ABB RAPID module: P41.mod

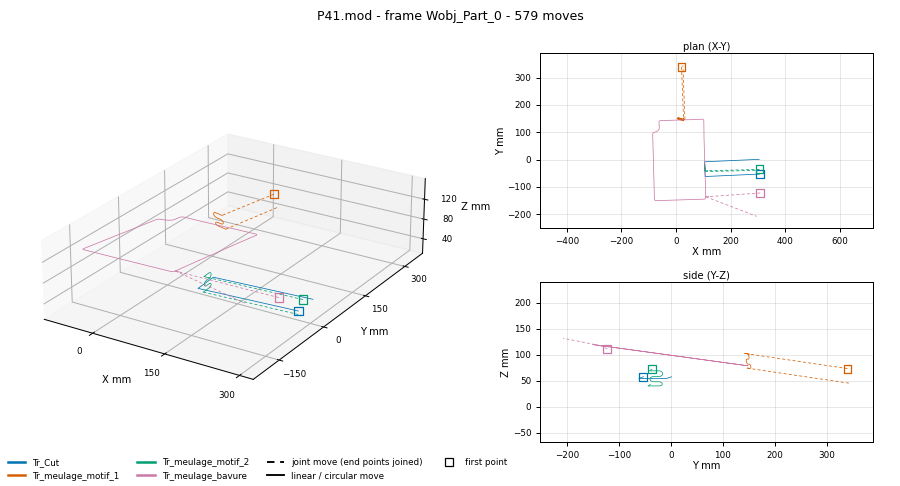
[picture p0: tool path of P41.mod in frame Wobj_Part_0, 579 of 588 moves have a stored position in this frame; points joined in program order, loops and branches not executed]
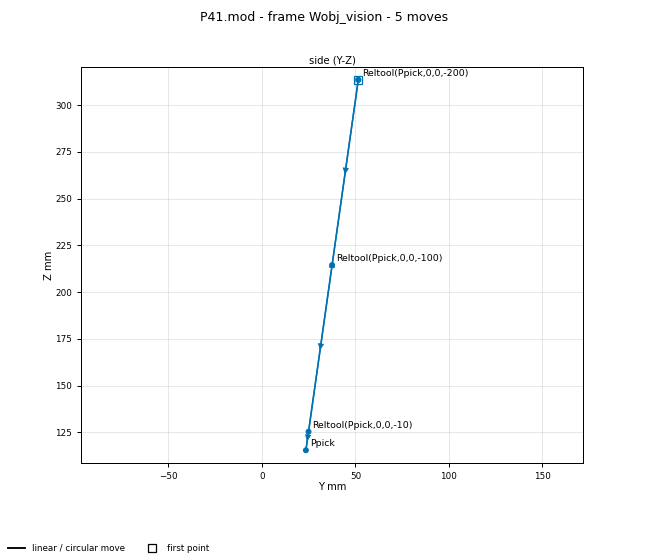
[picture p1: tool path of P41.mod in frame Wobj_vision, 5 of 588 moves have a stored position in this frame; points joined in program order, loops and branches not executed]
MODULE P41
	LOCAL CONST Speeddata vitesse_Tronconnage :=[10, 500, 0, 0];
	LOCAL CONST Robtarget Coupe_0 :=[[105.2163046875,-29.7869296875,54.5294296875],[0.0104555272873827,0.0212605825828778,-0.706787087904297,-0.707029477425901],[0,0,0,0],[8.999999E+09,8.999999E+09,8.999999E+09,8.999999E+09,8.999999E+09,8.999999E+09]];
	LOCAL CONST Robtarget Tr_meulage_motif_1_App1 :=[[20.0512236789454,339.562295836737,73.4032374615753],[0.0144291641931026,-0.0124615274841837,0.653500364086891,-0.756686053586129],[0,0,0,0],[8.999999E+09,8.999999E+09,8.999999E+09,8.999999E+09,8.999999E+09,8.999999E+09]];
	LOCAL CONST Robtarget Tr_meulage_motif_1_App2 :=[[27.2176163597285,151.722671041837,101.060391560579],[0.0144291641931026,-0.0124615274841837,0.653500364086891,-0.756686053586129],[0,0,0,0],[8.999999E+09,8.999999E+09,8.999999E+09,8.999999E+09,8.999999E+09,8.999999E+09]];
	LOCAL CONST Robtarget Tr_meulage_motif_1_P0 :=[[27.594794921875,141.836375,102.51603125],[0.0144291641931026,-0.0124615274841837,0.653500364086891,-0.756686053586129],[0,0,0,0],[8.999999E+09,8.999999E+09,8.999999E+09,8.999999E+09,8.999999E+09,8.999999E+09]];
	LOCAL CONST Robtarget Tr_meulage_motif_1_P1 :=[[26.6349609375,142.116578125,102.5018671875],[0.0144291641931026,-0.0124615274841837,0.653500364086891,-0.756686053586129],[0,0,0,0],[8.999999E+09,8.999999E+09,8.999999E+09,8.999999E+09,8.999999E+09,8.999999E+09]];
	LOCAL CONST Robtarget Tr_meulage_motif_1_P2 :=[[25.675126953125,142.396796875,102.487703125],[0.0144291641931026,-0.0124615274841837,0.653500364086891,-0.756686053586129],[0,0,0,0],[8.999999E+09,8.999999E+09,8.999999E+09,8.999999E+09,8.999999E+09,8.999999E+09]];
	LOCAL CONST Robtarget Tr_meulage_motif_1_P3 :=[[24.71529296875,142.677,102.4735390625],[0.0144291641931026,-0.0124615274841837,0.653500364086891,-0.756686053586129],[0,0,0,0],[8.999999E+09,8.999999E+09,8.999999E+09,8.999999E+09,8.999999E+09,8.999999E+09]];
	LOCAL CONST Robtarget Tr_meulage_motif_1_P4 :=[[23.755458984375,142.95721875,102.4593671875],[0.0144291641931026,-0.0124615274841837,0.653500364086891,-0.756686053586129],[0,0,0,0],[8.999999E+09,8.999999E+09,8.999999E+09,8.999999E+09,8.999999E+09,8.999999E+09]];
	LOCAL CONST Robtarget Tr_meulage_motif_1_P5 :=[[22.795625,143.237421875,102.445203125],[0.0144291641931026,-0.0124615274841837,0.653500364086891,-0.756686053586129],[0,0,0,0],[8.999999E+09,8.999999E+09,8.999999E+09,8.999999E+09,8.999999E+09,8.999999E+09]];
	LOCAL CONST Robtarget Tr_meulage_motif_1_P6 :=[[21.835791015625,143.517640625,102.4310390625],[0.0144291641931026,-0.0124615274841837,0.653500364086891,-0.756686053586129],[0,0,0,0],[8.999999E+09,8.999999E+09,8.999999E+09,8.999999E+09,8.999999E+09,8.999999E+09]];
	LOCAL CONST Robtarget Tr_meulage_motif_1_P7 :=[[20.87595703125,143.79784375,102.416875],[0.0144291641931026,-0.0124615274841837,0.653500364086891,-0.756686053586129],[0,0,0,0],[8.999999E+09,8.999999E+09,8.999999E+09,8.999999E+09,8.999999E+09,8.999999E+09]];
	LOCAL CONST Robtarget Tr_meulage_motif_1_P8 :=[[19.916123046875,144.0780625,102.4027109375],[0.0144291641931026,-0.0124615274841837,0.653500364086891,-0.756686053586129],[0,0,0,0],[8.999999E+09,8.999999E+09,8.999999E+09,8.999999E+09,8.999999E+09,8.999999E+09]];
	LOCAL CONST Robtarget Tr_meulage_motif_1_P9 :=[[18.9562890625,144.358265625,102.3885390625],[0.0144291641931026,-0.0124615274841837,0.653500364086891,-0.756686053586129],[0,0,0,0],[8.999999E+09,8.999999E+09,8.999999E+09,8.999999E+09,8.999999E+09,8.999999E+09]];
	LOCAL CONST Robtarget Tr_meulage_motif_1_P10 :=[[17.99645703125,144.638484375,102.374375],[0.0144291641931026,-0.0124615274841837,0.653500364086891,-0.756686053586129],[0,0,0,0],[8.999999E+09,8.999999E+09,8.999999E+09,8.999999E+09,8.999999E+09,8.999999E+09]];
	LOCAL CONST Robtarget Tr_meulage_motif_1_P11 :=[[17.036623046875,144.9186875,102.3602109375],[0.0144291641931026,-0.0124615274841837,0.653500364086891,-0.756686053586129],[0,0,0,0],[8.999999E+09,8.999999E+09,8.999999E+09,8.999999E+09,8.999999E+09,8.999999E+09]];
	LOCAL CONST Robtarget Tr_meulage_motif_1_P12 :=[[16.0767880859375,145.19890625,102.346046875],[0.0144291641931026,-0.0124615274841837,0.653500364086891,-0.756686053586129],[0,0,0,0],[8.999999E+09,8.999999E+09,8.999999E+09,8.999999E+09,8.999999E+09,8.999999E+09]];
	LOCAL CONST Robtarget Tr_meulage_motif_1_P13 :=[[15.116955078125,145.479109375,102.331875],[0.0144291641931026,-0.0124615274841837,0.653500364086891,-0.756686053586129],[0,0,0,0],[8.999999E+09,8.999999E+09,8.999999E+09,8.999999E+09,8.999999E+09,8.999999E+09]];
	LOCAL CONST Robtarget Tr_meulage_motif_1_P14 :=[[14.15712109375,145.759328125,102.3177109375],[0.0144291641931026,-0.0124615274841837,0.653500364086891,-0.756686053586129],[0,0,0,0],[8.999999E+09,8.999999E+09,8.999999E+09,8.999999E+09,8.999999E+09,8.999999E+09]];
	LOCAL CONST Robtarget Tr_meulage_motif_1_P15 :=[[13.197287109375,146.03953125,102.303546875],[0.0144291641931026,-0.0124615274841837,0.653500364086891,-0.756686053586129],[0,0,0,0],[8.999999E+09,8.999999E+09,8.999999E+09,8.999999E+09,8.999999E+09,8.999999E+09]];
	LOCAL CONST Robtarget Tr_meulage_motif_1_P16 :=[[12.237453125,146.31975,102.2893828125],[0.0144291641931026,-0.0124615274841837,0.653500364086891,-0.756686053586129],[0,0,0,0],[8.999999E+09,8.999999E+09,8.999999E+09,8.999999E+09,8.999999E+09,8.999999E+09]];
	LOCAL CONST Robtarget Tr_meulage_motif_1_P17 :=[[11.277619140625,146.59996875,102.27521875],[0.0144291641931026,-0.0124615274841837,0.653500364086891,-0.756686053586129],[0,0,0,0],[8.999999E+09,8.999999E+09,8.999999E+09,8.999999E+09,8.999999E+09,8.999999E+09]];
	LOCAL CONST Robtarget Tr_meulage_motif_1_P18 :=[[10.31778515625,146.880171875,102.261046875],[0.0144291641931026,-0.0124615274841837,0.653500364086891,-0.756686053586129],[0,0,0,0],[8.999999E+09,8.999999E+09,8.999999E+09,8.999999E+09,8.999999E+09,8.999999E+09]];
	LOCAL CONST Robtarget Tr_meulage_motif_1_P19 :=[[9.3730380859375,147.1800625,102.1388515625],[0.0144291641931026,-0.0124615274841837,0.653500364086891,-0.756686053586129],[0,0,0,0],[8.999999E+09,8.999999E+09,8.999999E+09,8.999999E+09,8.999999E+09,8.999999E+09]];
	LOCAL CONST Robtarget Tr_meulage_motif_1_P20 :=[[8.4797333984375,147.486828125,101.9189375],[0.0144291641931026,-0.0124615274841837,0.653500364086891,-0.756686053586129],[0,0,0,0],[8.999999E+09,8.999999E+09,8.999999E+09,8.999999E+09,8.999999E+09,8.999999E+09]];
	LOCAL CONST Robtarget Tr_meulage_motif_1_P21 :=[[7.68080224609375,147.77925,101.641046875],[0.0144291641931026,-0.0124615274841837,0.653500364086891,-0.756686053586129],[0,0,0,0],[8.999999E+09,8.999999E+09,8.999999E+09,8.999999E+09,8.999999E+09,8.999999E+09]];
	LOCAL CONST Robtarget Tr_meulage_motif_1_P22 :=[[6.98081787109375,148.0436875,101.3606015625],[0.0144291641931026,-0.0124615274841837,0.653500364086891,-0.756686053586129],[0,0,0,0],[8.999999E+09,8.999999E+09,8.999999E+09,8.999999E+09,8.999999E+09,8.999999E+09]];
	LOCAL CONST Robtarget Tr_meulage_motif_1_P23 :=[[5.96826025390625,148.4734375,100.742546875],[0.0144291641931026,-0.0124615274841837,0.653500364086891,-0.756686053586129],[0,0,0,0],[8.999999E+09,8.999999E+09,8.999999E+09,8.999999E+09,8.999999E+09,8.999999E+09]];
	LOCAL CONST Robtarget Tr_meulage_motif_1_P24 :=[[5.0464296875,148.927109375,99.8991953125],[0.0144291641931026,-0.0124615274841837,0.653500364086891,-0.756686053586129],[0,0,0,0],[8.999999E+09,8.999999E+09,8.999999E+09,8.999999E+09,8.999999E+09,8.999999E+09]];
	LOCAL CONST Robtarget Tr_meulage_motif_1_P25 :=[[4.30640478515625,149.3660625,98.8860234375],[0.0144291641931026,-0.0124615274841837,0.653500364086891,-0.756686053586129],[0,0,0,0],[8.999999E+09,8.999999E+09,8.999999E+09,8.999999E+09,8.999999E+09,8.999999E+09]];
	LOCAL CONST Robtarget Tr_meulage_motif_1_P26 :=[[3.91807373046875,149.722453125,97.7876796875],[0.0144291641931026,-0.0124615274841837,0.653500364086891,-0.756686053586129],[0,0,0,0],[8.999999E+09,8.999999E+09,8.999999E+09,8.999999E+09,8.999999E+09,8.999999E+09]];
	LOCAL CONST Robtarget Tr_meulage_motif_1_P27 :=[[3.9421162109375,149.86696875,97.106765625],[0.0144291641931026,-0.0124615274841837,0.653500364086891,-0.756686053586129],[0,0,0,0],[8.999999E+09,8.999999E+09,8.999999E+09,8.999999E+09,8.999999E+09,8.999999E+09]];
	LOCAL CONST Robtarget Tr_meulage_motif_1_P28 :=[[3.98963891601562,149.9970625,96.4601875],[0.0144291641931026,-0.0124615274841837,0.653500364086891,-0.756686053586129],[0,0,0,0],[8.999999E+09,8.999999E+09,8.999999E+09,8.999999E+09,8.999999E+09,8.999999E+09]];
	LOCAL CONST Robtarget Tr_meulage_motif_1_P29 :=[[4.0898212890625,150.11175,95.81453125],[0.0144291641931026,-0.0124615274841837,0.653500364086891,-0.756686053586129],[0,0,0,0],[8.999999E+09,8.999999E+09,8.999999E+09,8.999999E+09,8.999999E+09,8.999999E+09]];
	LOCAL CONST Robtarget Tr_meulage_motif_1_P30 :=[[4.647208984375,150.18890625,94.74428125],[0.0144291641931026,-0.0124615274841837,0.653500364086891,-0.756686053586129],[0,0,0,0],[8.999999E+09,8.999999E+09,8.999999E+09,8.999999E+09,8.999999E+09,8.999999E+09]];
	LOCAL CONST Robtarget Tr_meulage_motif_1_P31 :=[[5.54177099609375,150.146921875,93.7721171875],[0.0144291641931026,-0.0124615274841837,0.653500364086891,-0.756686053586129],[0,0,0,0],[8.999999E+09,8.999999E+09,8.999999E+09,8.999999E+09,8.999999E+09,8.999999E+09]];
	LOCAL CONST Robtarget Tr_meulage_motif_1_P32 :=[[6.583640625,150.023234375,92.976125],[0.0144291641931026,-0.0124615274841837,0.653500364086891,-0.756686053586129],[0,0,0,0],[8.999999E+09,8.999999E+09,8.999999E+09,8.999999E+09,8.999999E+09,8.999999E+09]];
	LOCAL CONST Robtarget Tr_meulage_motif_1_P33 :=[[7.271578125,149.9085625,92.598890625],[0.0144291641931026,-0.0124615274841837,0.653500364086891,-0.756686053586129],[0,0,0,0],[8.999999E+09,8.999999E+09,8.999999E+09,8.999999E+09,8.999999E+09,8.999999E+09]];
	LOCAL CONST Robtarget Tr_meulage_motif_1_P34 :=[[8.41825390625,149.679953125,92.138578125],[0.0144291641931026,-0.0124615274841837,0.653500364086891,-0.756686053586129],[0,0,0,0],[8.999999E+09,8.999999E+09,8.999999E+09,8.999999E+09,8.999999E+09,8.999999E+09]];
	LOCAL CONST Robtarget Tr_meulage_motif_1_P35 :=[[9.2483232421875,149.495125,91.8923125],[0.0144291641931026,-0.0124615274841837,0.653500364086891,-0.756686053586129],[0,0,0,0],[8.999999E+09,8.999999E+09,8.999999E+09,8.999999E+09,8.999999E+09,8.999999E+09]];
	LOCAL CONST Robtarget Tr_meulage_motif_1_P36 :=[[10.1575830078125,149.2741875,91.7055859375],[0.0144291641931026,-0.0124615274841837,0.653500364086891,-0.756686053586129],[0,0,0,0],[8.999999E+09,8.999999E+09,8.999999E+09,8.999999E+09,8.999999E+09,8.999999E+09]];
	LOCAL CONST Robtarget Tr_meulage_motif_1_P37 :=[[11.1075244140625,149.020515625,91.6133046875],[0.0144291641931026,-0.0124615274841837,0.653500364086891,-0.756686053586129],[0,0,0,0],[8.999999E+09,8.999999E+09,8.999999E+09,8.999999E+09,8.999999E+09,8.999999E+09]];
	LOCAL CONST Robtarget Tr_meulage_motif_1_P38 :=[[12.0681669921875,148.764140625,91.5192265625],[0.0144291641931026,-0.0124615274841837,0.653500364086891,-0.756686053586129],[0,0,0,0],[8.999999E+09,8.999999E+09,8.999999E+09,8.999999E+09,8.999999E+09,8.999999E+09]];
	LOCAL CONST Robtarget Tr_meulage_motif_1_P39 :=[[13.0280009765625,148.4839375,91.533390625],[0.0144291641931026,-0.0124615274841837,0.653500364086891,-0.756686053586129],[0,0,0,0],[8.999999E+09,8.999999E+09,8.999999E+09,8.999999E+09,8.999999E+09,8.999999E+09]];
	LOCAL CONST Robtarget Tr_meulage_motif_1_P40 :=[[13.9878349609375,148.20371875,91.5475546875],[0.0144291641931026,-0.0124615274841837,0.653500364086891,-0.756686053586129],[0,0,0,0],[8.999999E+09,8.999999E+09,8.999999E+09,8.999999E+09,8.999999E+09,8.999999E+09]];
	LOCAL CONST Robtarget Tr_meulage_motif_1_P41 :=[[14.9476689453125,147.9235,91.56171875],[0.0144291641931026,-0.0124615274841837,0.653500364086891,-0.756686053586129],[0,0,0,0],[8.999999E+09,8.999999E+09,8.999999E+09,8.999999E+09,8.999999E+09,8.999999E+09]];
	LOCAL CONST Robtarget Tr_meulage_motif_1_P42 :=[[15.9075029296875,147.643296875,91.575890625],[0.0144291641931026,-0.0124615274841837,0.653500364086891,-0.756686053586129],[0,0,0,0],[8.999999E+09,8.999999E+09,8.999999E+09,8.999999E+09,8.999999E+09,8.999999E+09]];
	LOCAL CONST Robtarget Tr_meulage_motif_1_P43 :=[[16.8673359375,147.363078125,91.5900546875],[0.0144291641931026,-0.0124615274841837,0.653500364086891,-0.756686053586129],[0,0,0,0],[8.999999E+09,8.999999E+09,8.999999E+09,8.999999E+09,8.999999E+09,8.999999E+09]];
	LOCAL CONST Robtarget Tr_meulage_motif_1_P44 :=[[17.827169921875,147.082875,91.60421875],[0.0144291641931026,-0.0124615274841837,0.653500364086891,-0.756686053586129],[0,0,0,0],[8.999999E+09,8.999999E+09,8.999999E+09,8.999999E+09,8.999999E+09,8.999999E+09]];
	LOCAL CONST Robtarget Tr_meulage_motif_1_P45 :=[[18.78700390625,146.80265625,91.6183828125],[0.0144291641931026,-0.0124615274841837,0.653500364086891,-0.756686053586129],[0,0,0,0],[8.999999E+09,8.999999E+09,8.999999E+09,8.999999E+09,8.999999E+09,8.999999E+09]];
	LOCAL CONST Robtarget Tr_meulage_motif_1_P46 :=[[19.746837890625,146.522453125,91.632546875],[0.0144291641931026,-0.0124615274841837,0.653500364086891,-0.756686053586129],[0,0,0,0],[8.999999E+09,8.999999E+09,8.999999E+09,8.999999E+09,8.999999E+09,8.999999E+09]];
	LOCAL CONST Robtarget Tr_meulage_motif_1_P47 :=[[20.706671875,146.242234375,91.64671875],[0.0144291641931026,-0.0124615274841837,0.653500364086891,-0.756686053586129],[0,0,0,0],[8.999999E+09,8.999999E+09,8.999999E+09,8.999999E+09,8.999999E+09,8.999999E+09]];
	LOCAL CONST Robtarget Tr_meulage_motif_1_P48 :=[[21.666505859375,145.96203125,91.6608828125],[0.0144291641931026,-0.0124615274841837,0.653500364086891,-0.756686053586129],[0,0,0,0],[8.999999E+09,8.999999E+09,8.999999E+09,8.999999E+09,8.999999E+09,8.999999E+09]];
	LOCAL CONST Robtarget Tr_meulage_motif_1_P49 :=[[22.6271484375,145.70565625,91.5668046875],[0.0144291641931026,-0.0124615274841837,0.653500364086891,-0.756686053586129],[0,0,0,0],[8.999999E+09,8.999999E+09,8.999999E+09,8.999999E+09,8.999999E+09,8.999999E+09]];
	LOCAL CONST Robtarget Tr_meulage_motif_1_P50 :=[[23.55080859375,145.481984375,91.373703125],[0.0144291641931026,-0.0124615274841837,0.653500364086891,-0.756686053586129],[0,0,0,0],[8.999999E+09,8.999999E+09,8.999999E+09,8.999999E+09,8.999999E+09,8.999999E+09]];
	LOCAL CONST Robtarget Tr_meulage_motif_1_P51 :=[[24.388814453125,145.29653125,91.11996875],[0.0144291641931026,-0.0124615274841837,0.653500364086891,-0.756686053586129],[0,0,0,0],[8.999999E+09,8.999999E+09,8.999999E+09,8.999999E+09,8.999999E+09,8.999999E+09]];
	LOCAL CONST Robtarget Tr_meulage_motif_1_P52 :=[[25.093595703125,145.157,90.832640625],[0.0144291641931026,-0.0124615274841837,0.653500364086891,-0.756686053586129],[0,0,0,0],[8.999999E+09,8.999999E+09,8.999999E+09,8.999999E+09,8.999999E+09,8.999999E+09]];
	LOCAL CONST Robtarget Tr_meulage_motif_1_P53 :=[[26.13412890625,144.997484375,90.1994609375],[0.0144291641931026,-0.0124615274841837,0.653500364086891,-0.756686053586129],[0,0,0,0],[8.999999E+09,8.999999E+09,8.999999E+09,8.999999E+09,8.999999E+09,8.999999E+09]];
	LOCAL CONST Robtarget Tr_meulage_motif_1_P54 :=[[27.064658203125,144.922203125,89.3303046875],[0.0144291641931026,-0.0124615274841837,0.653500364086891,-0.756686053586129],[0,0,0,0],[8.999999E+09,8.999999E+09,8.999999E+09,8.999999E+09,8.999999E+09,8.999999E+09]];
	LOCAL CONST Robtarget Tr_meulage_motif_1_P55 :=[[27.65331640625,144.97809375,88.3150625],[0.0144291641931026,-0.0124615274841837,0.653500364086891,-0.756686053586129],[0,0,0,0],[8.999999E+09,8.999999E+09,8.999999E+09,8.999999E+09,8.999999E+09,8.999999E+09]];
	LOCAL CONST Robtarget Tr_meulage_motif_1_P56 :=[[27.88049609375,145.062703125,87.6398359375],[0.0144291641931026,-0.0124615274841837,0.653500364086891,-0.756686053586129],[0,0,0,0],[8.999999E+09,8.999999E+09,8.999999E+09,8.999999E+09,8.999999E+09,8.999999E+09]];
	LOCAL CONST Robtarget Tr_meulage_motif_1_P57 :=[[27.99711328125,145.1963125,86.8878203125],[0.0144291641931026,-0.0124615274841837,0.653500364086891,-0.756686053586129],[0,0,0,0],[8.999999E+09,8.999999E+09,8.999999E+09,8.999999E+09,8.999999E+09,8.999999E+09]];
	LOCAL CONST Robtarget Tr_meulage_motif_1_P58 :=[[27.988193359375,145.36653125,86.134078125],[0.0144291641931026,-0.0124615274841837,0.653500364086891,-0.756686053586129],[0,0,0,0],[8.999999E+09,8.999999E+09,8.999999E+09,8.999999E+09,8.999999E+09,8.999999E+09]];
	LOCAL CONST Robtarget Tr_meulage_motif_1_P59 :=[[27.6651015625,145.702140625,85.0444609375],[0.0144291641931026,-0.0124615274841837,0.653500364086891,-0.756686053586129],[0,0,0,0],[8.999999E+09,8.999999E+09,8.999999E+09,8.999999E+09,8.999999E+09,8.999999E+09]];
	LOCAL CONST Robtarget Tr_meulage_motif_1_P60 :=[[27.309521484375,145.93346875,84.4658984375],[0.0144291641931026,-0.0124615274841837,0.653500364086891,-0.756686053586129],[0,0,0,0],[8.999999E+09,8.999999E+09,8.999999E+09,8.999999E+09,8.999999E+09,8.999999E+09]];
	LOCAL CONST Robtarget Tr_meulage_motif_1_P61 :=[[26.52178515625,146.35659375,83.585890625],[0.0144291641931026,-0.0124615274841837,0.653500364086891,-0.756686053586129],[0,0,0,0],[8.999999E+09,8.999999E+09,8.999999E+09,8.999999E+09,8.999999E+09,8.999999E+09]];
	LOCAL CONST Robtarget Tr_meulage_motif_1_P62 :=[[25.9893984375,146.60221875,83.17246875],[0.0144291641931026,-0.0124615274841837,0.653500364086891,-0.756686053586129],[0,0,0,0],[8.999999E+09,8.999999E+09,8.999999E+09,8.999999E+09,8.999999E+09,8.999999E+09]];
	LOCAL CONST Robtarget Tr_meulage_motif_1_P63 :=[[24.955498046875,147.022515625,82.624609375],[0.0144291641931026,-0.0124615274841837,0.653500364086891,-0.756686053586129],[0,0,0,0],[8.999999E+09,8.999999E+09,8.999999E+09,8.999999E+09,8.999999E+09,8.999999E+09]];
	LOCAL CONST Robtarget Tr_meulage_motif_1_P64 :=[[24.18430078125,147.312,82.32396875],[0.0144291641931026,-0.0124615274841837,0.653500364086891,-0.756686053586129],[0,0,0,0],[8.999999E+09,8.999999E+09,8.999999E+09,8.999999E+09,8.999999E+09,8.999999E+09]];
	LOCAL CONST Robtarget Tr_meulage_motif_1_P65 :=[[23.304431640625,147.613375,82.110828125],[0.0144291641931026,-0.0124615274841837,0.653500364086891,-0.756686053586129],[0,0,0,0],[8.999999E+09,8.999999E+09,8.999999E+09,8.999999E+09,8.999999E+09,8.999999E+09]];
	LOCAL CONST Robtarget Tr_meulage_motif_1_P66 :=[[22.370099609375,147.909796875,81.9907421875],[0.0144291641931026,-0.0124615274841837,0.653500364086891,-0.756686053586129],[0,0,0,0],[8.999999E+09,8.999999E+09,8.999999E+09,8.999999E+09,8.999999E+09,8.999999E+09]];
	LOCAL CONST Robtarget Tr_meulage_motif_1_P67 :=[[21.4253515625,148.209671875,81.8685390625],[0.0144291641931026,-0.0124615274841837,0.653500364086891,-0.756686053586129],[0,0,0,0],[8.999999E+09,8.999999E+09,8.999999E+09,8.999999E+09,8.999999E+09,8.999999E+09]];
	LOCAL CONST Robtarget Tr_meulage_motif_1_P68 :=[[20.465517578125,148.489890625,81.854375],[0.0144291641931026,-0.0124615274841837,0.653500364086891,-0.756686053586129],[0,0,0,0],[8.999999E+09,8.999999E+09,8.999999E+09,8.999999E+09,8.999999E+09,8.999999E+09]];
	LOCAL CONST Robtarget Tr_meulage_motif_1_P69 :=[[19.50568359375,148.77009375,81.8402109375],[0.0144291641931026,-0.0124615274841837,0.653500364086891,-0.756686053586129],[0,0,0,0],[8.999999E+09,8.999999E+09,8.999999E+09,8.999999E+09,8.999999E+09,8.999999E+09]];
	LOCAL CONST Robtarget Tr_meulage_motif_1_P70 :=[[18.545849609375,149.0503125,81.826046875],[0.0144291641931026,-0.0124615274841837,0.653500364086891,-0.756686053586129],[0,0,0,0],[8.999999E+09,8.999999E+09,8.999999E+09,8.999999E+09,8.999999E+09,8.999999E+09]];
	LOCAL CONST Robtarget Tr_meulage_motif_1_P71 :=[[17.586015625,149.330515625,81.811875],[0.0144291641931026,-0.0124615274841837,0.653500364086891,-0.756686053586129],[0,0,0,0],[8.999999E+09,8.999999E+09,8.999999E+09,8.999999E+09,8.999999E+09,8.999999E+09]];
	LOCAL CONST Robtarget Tr_meulage_motif_1_P72 :=[[16.62618359375,149.610734375,81.7977109375],[0.0144291641931026,-0.0124615274841837,0.653500364086891,-0.756686053586129],[0,0,0,0],[8.999999E+09,8.999999E+09,8.999999E+09,8.999999E+09,8.999999E+09,8.999999E+09]];
	LOCAL CONST Robtarget Tr_meulage_motif_1_P73 :=[[15.6663486328125,149.8909375,81.783546875],[0.0144291641931026,-0.0124615274841837,0.653500364086891,-0.756686053586129],[0,0,0,0],[8.999999E+09,8.999999E+09,8.999999E+09,8.999999E+09,8.999999E+09,8.999999E+09]];
	LOCAL CONST Robtarget Tr_meulage_motif_1_P74 :=[[14.7065146484375,150.17115625,81.7693828125],[0.0144291641931026,-0.0124615274841837,0.653500364086891,-0.756686053586129],[0,0,0,0],[8.999999E+09,8.999999E+09,8.999999E+09,8.999999E+09,8.999999E+09,8.999999E+09]];
	LOCAL CONST Robtarget Tr_meulage_motif_1_P75 :=[[13.746681640625,150.451359375,81.75521875],[0.0144291641931026,-0.0124615274841837,0.653500364086891,-0.756686053586129],[0,0,0,0],[8.999999E+09,8.999999E+09,8.999999E+09,8.999999E+09,8.999999E+09,8.999999E+09]];
	LOCAL CONST Robtarget Tr_meulage_motif_1_P76 :=[[12.78684765625,150.731578125,81.741046875],[0.0144291641931026,-0.0124615274841837,0.653500364086891,-0.756686053586129],[0,0,0,0],[8.999999E+09,8.999999E+09,8.999999E+09,8.999999E+09,8.999999E+09,8.999999E+09]];
	LOCAL CONST Robtarget Tr_meulage_motif_1_P77 :=[[11.827013671875,151.01178125,81.7268828125],[0.0144291641931026,-0.0124615274841837,0.653500364086891,-0.756686053586129],[0,0,0,0],[8.999999E+09,8.999999E+09,8.999999E+09,8.999999E+09,8.999999E+09,8.999999E+09]];
	LOCAL CONST Robtarget Tr_meulage_motif_1_P78 :=[[10.8822666015625,151.311671875,81.6046796875],[0.0144291641931026,-0.0124615274841837,0.653500364086891,-0.756686053586129],[0,0,0,0],[8.999999E+09,8.999999E+09,8.999999E+09,8.999999E+09,8.999999E+09,8.999999E+09]];
	LOCAL CONST Robtarget Tr_meulage_motif_1_P79 :=[[9.9889619140625,151.6184375,81.3847734375],[0.0144291641931026,-0.0124615274841837,0.653500364086891,-0.756686053586129],[0,0,0,0],[8.999999E+09,8.999999E+09,8.999999E+09,8.999999E+09,8.999999E+09,8.999999E+09]];
	LOCAL CONST Robtarget Tr_meulage_motif_1_P80 :=[[9.1900302734375,151.910875,81.106875],[0.0144291641931026,-0.0124615274841837,0.653500364086891,-0.756686053586129],[0,0,0,0],[8.999999E+09,8.999999E+09,8.999999E+09,8.999999E+09,8.999999E+09,8.999999E+09]];
	LOCAL CONST Robtarget Tr_meulage_motif_1_P81 :=[[8.4900458984375,152.175296875,80.8264375],[0.0144291641931026,-0.0124615274841837,0.653500364086891,-0.756686053586129],[0,0,0,0],[8.999999E+09,8.999999E+09,8.999999E+09,8.999999E+09,8.999999E+09,8.999999E+09]];
	LOCAL CONST Robtarget Tr_meulage_motif_1_P82 :=[[7.47748828125,152.605046875,80.2083828125],[0.0144291641931026,-0.0124615274841837,0.653500364086891,-0.756686053586129],[0,0,0,0],[8.999999E+09,8.999999E+09,8.999999E+09,8.999999E+09,8.999999E+09,8.999999E+09]];
	LOCAL CONST Robtarget Tr_meulage_motif_1_P83 :=[[6.6234453125,153.049015625,79.3206953125],[0.0144291641931026,-0.0124615274841837,0.653500364086891,-0.756686053586129],[0,0,0,0],[8.999999E+09,8.999999E+09,8.999999E+09,8.999999E+09,8.999999E+09,8.999999E+09]];
	LOCAL CONST Robtarget Tr_meulage_motif_1_P84 :=[[6.1168349609375,153.433359375,78.25015625],[0.0144291641931026,-0.0124615274841837,0.653500364086891,-0.756686053586129],[0,0,0,0],[8.999999E+09,8.999999E+09,8.999999E+09,8.999999E+09,8.999999E+09,8.999999E+09]];
	LOCAL CONST Robtarget Tr_meulage_motif_1_P85 :=[[6.025068359375,153.67446875,77.28521875],[0.0144291641931026,-0.0124615274841837,0.653500364086891,-0.756686053586129],[0,0,0,0],[8.999999E+09,8.999999E+09,8.999999E+09,8.999999E+09,8.999999E+09,8.999999E+09]];
	LOCAL CONST Robtarget Tr_meulage_motif_1_P86 :=[[6.16596484375,153.67790625,77.0869609375],[0.0144291641931026,-0.0124615274841837,0.653500364086891,-0.756686053586129],[0,0,0,0],[8.999999E+09,8.999999E+09,8.999999E+09,8.999999E+09,8.999999E+09,8.999999E+09]];
	LOCAL CONST Robtarget Tr_meulage_motif_1_P87 :=[[6.33658935546875,153.78625,76.3784140625],[0.0144291641931026,-0.0124615274841837,0.653500364086891,-0.756686053586129],[0,0,0,0],[8.999999E+09,8.999999E+09,8.999999E+09,8.999999E+09,8.999999E+09,8.999999E+09]];
	LOCAL CONST Robtarget Tr_meulage_motif_1_P88 :=[[7.06044921875,153.77890625,75.471984375],[0.0144291641931026,-0.0124615274841837,0.653500364086891,-0.756686053586129],[0,0,0,0],[8.999999E+09,8.999999E+09,8.999999E+09,8.999999E+09,8.999999E+09,8.999999E+09]];
	LOCAL CONST Robtarget Tr_meulage_motif_1_P89 :=[[7.62901025390625,153.71390625,75.026359375],[0.0144291641931026,-0.0124615274841837,0.653500364086891,-0.756686053586129],[0,0,0,0],[8.999999E+09,8.999999E+09,8.999999E+09,8.999999E+09,8.999999E+09,8.999999E+09]];
	LOCAL CONST Robtarget Tr_meulage_motif_1_P90 :=[[8.7520439453125,153.501546875,74.523703125],[0.0144291641931026,-0.0124615274841837,0.653500364086891,-0.756686053586129],[0,0,0,0],[8.999999E+09,8.999999E+09,8.999999E+09,8.999999E+09,8.999999E+09,8.999999E+09]];
	LOCAL CONST Robtarget Tr_meulage_motif_1_P91 :=[[9.58211328125,153.31671875,74.2774375],[0.0144291641931026,-0.0124615274841837,0.653500364086891,-0.756686053586129],[0,0,0,0],[8.999999E+09,8.999999E+09,8.999999E+09,8.999999E+09,8.999999E+09,8.999999E+09]];
	LOCAL CONST Robtarget Tr_meulage_motif_1_P92 :=[[10.491373046875,153.09578125,74.090703125],[0.0144291641931026,-0.0124615274841837,0.653500364086891,-0.756686053586129],[0,0,0,0],[8.999999E+09,8.999999E+09,8.999999E+09,8.999999E+09,8.999999E+09,8.999999E+09]];
	LOCAL CONST Robtarget Tr_meulage_motif_1_P93 :=[[11.441314453125,152.842109375,73.998421875],[0.0144291641931026,-0.0124615274841837,0.653500364086891,-0.756686053586129],[0,0,0,0],[8.999999E+09,8.999999E+09,8.999999E+09,8.999999E+09,8.999999E+09,8.999999E+09]];
	LOCAL CONST Robtarget Tr_meulage_motif_1_P94 :=[[12.4019580078125,152.585734375,73.90434375],[0.0144291641931026,-0.0124615274841837,0.653500364086891,-0.756686053586129],[0,0,0,0],[8.999999E+09,8.999999E+09,8.999999E+09,8.999999E+09,8.999999E+09,8.999999E+09]];
	LOCAL CONST Robtarget Tr_meulage_motif_1_P95 :=[[13.361791015625,152.30553125,73.9185078125],[0.0144291641931026,-0.0124615274841837,0.653500364086891,-0.756686053586129],[0,0,0,0],[8.999999E+09,8.999999E+09,8.999999E+09,8.999999E+09,8.999999E+09,8.999999E+09]];
	LOCAL CONST Robtarget Tr_meulage_motif_1_P96 :=[[14.321625,152.0253125,73.932671875],[0.0144291641931026,-0.0124615274841837,0.653500364086891,-0.756686053586129],[0,0,0,0],[8.999999E+09,8.999999E+09,8.999999E+09,8.999999E+09,8.999999E+09,8.999999E+09]];
	LOCAL CONST Robtarget Tr_meulage_motif_1_P97 :=[[15.281458984375,151.745109375,73.94684375],[0.0144291641931026,-0.0124615274841837,0.653500364086891,-0.756686053586129],[0,0,0,0],[8.999999E+09,8.999999E+09,8.999999E+09,8.999999E+09,8.999999E+09,8.999999E+09]];
	LOCAL CONST Robtarget Tr_meulage_motif_1_P98 :=[[16.24129296875,151.464890625,73.9610078125],[0.0144291641931026,-0.0124615274841837,0.653500364086891,-0.756686053586129],[0,0,0,0],[8.999999E+09,8.999999E+09,8.999999E+09,8.999999E+09,8.999999E+09,8.999999E+09]];
	LOCAL CONST Robtarget Tr_meulage_motif_1_P99 :=[[17.201126953125,151.1846875,73.975171875],[0.0144291641931026,-0.0124615274841837,0.653500364086891,-0.756686053586129],[0,0,0,0],[8.999999E+09,8.999999E+09,8.999999E+09,8.999999E+09,8.999999E+09,8.999999E+09]];
	LOCAL CONST Robtarget Tr_meulage_motif_1_P100 :=[[18.1609609375,150.90446875,73.9893359375],[0.0144291641931026,-0.0124615274841837,0.653500364086891,-0.756686053586129],[0,0,0,0],[8.999999E+09,8.999999E+09,8.999999E+09,8.999999E+09,8.999999E+09,8.999999E+09]];
	LOCAL CONST Robtarget Tr_meulage_motif_1_P101 :=[[19.120794921875,150.624265625,74.0035078125],[0.0144291641931026,-0.0124615274841837,0.653500364086891,-0.756686053586129],[0,0,0,0],[8.999999E+09,8.999999E+09,8.999999E+09,8.999999E+09,8.999999E+09,8.999999E+09]];
	LOCAL CONST Robtarget Tr_meulage_motif_1_P102 :=[[20.08062890625,150.344046875,74.017671875],[0.0144291641931026,-0.0124615274841837,0.653500364086891,-0.756686053586129],[0,0,0,0],[8.999999E+09,8.999999E+09,8.999999E+09,8.999999E+09,8.999999E+09,8.999999E+09]];
	LOCAL CONST Robtarget Tr_meulage_motif_1_P103 :=[[21.040462890625,150.06384375,74.0318359375],[0.0144291641931026,-0.0124615274841837,0.653500364086891,-0.756686053586129],[0,0,0,0],[8.999999E+09,8.999999E+09,8.999999E+09,8.999999E+09,8.999999E+09,8.999999E+09]];
	LOCAL CONST Robtarget Tr_meulage_motif_1_P104 :=[[22.000294921875,149.783625,74.046],[0.0144291641931026,-0.0124615274841837,0.653500364086891,-0.756686053586129],[0,0,0,0],[8.999999E+09,8.999999E+09,8.999999E+09,8.999999E+09,8.999999E+09,8.999999E+09]];
	LOCAL CONST Robtarget Tr_meulage_motif_1_P105 :=[[22.96012890625,149.50340625,74.0601640625],[0.0144291641931026,-0.0124615274841837,0.653500364086891,-0.756686053586129],[0,0,0,0],[8.999999E+09,8.999999E+09,8.999999E+09,8.999999E+09,8.999999E+09,8.999999E+09]];
	LOCAL CONST Robtarget Tr_meulage_motif_1_P106 :=[[23.919962890625,149.223203125,74.0743359375],[0.0144291641931026,-0.0124615274841837,0.653500364086891,-0.756686053586129],[0,0,0,0],[8.999999E+09,8.999999E+09,8.999999E+09,8.999999E+09,8.999999E+09,8.999999E+09]];
	LOCAL CONST Robtarget Tr_meulage_motif_1_P107 :=[[24.879796875,148.942984375,74.0885],[0.0144291641931026,-0.0124615274841837,0.653500364086891,-0.756686053586129],[0,0,0,0],[8.999999E+09,8.999999E+09,8.999999E+09,8.999999E+09,8.999999E+09,8.999999E+09]];
	LOCAL CONST Robtarget Tr_meulage_motif_1_P108 :=[[25.839630859375,148.66278125,74.1026640625],[0.0144291641931026,-0.0124615274841837,0.653500364086891,-0.756686053586129],[0,0,0,0],[8.999999E+09,8.999999E+09,8.999999E+09,8.999999E+09,8.999999E+09,8.999999E+09]];
	LOCAL CONST Robtarget Tr_meulage_motif_1_P109 :=[[26.79946484375,148.3825625,74.116828125],[0.0144291641931026,-0.0124615274841837,0.653500364086891,-0.756686053586129],[0,0,0,0],[8.999999E+09,8.999999E+09,8.999999E+09,8.999999E+09,8.999999E+09,8.999999E+09]];
	LOCAL CONST Robtarget Tr_meulage_motif_1_P110 :=[[27.759298828125,148.102359375,74.131],[0.0144291641931026,-0.0124615274841837,0.653500364086891,-0.756686053586129],[0,0,0,0],[8.999999E+09,8.999999E+09,8.999999E+09,8.999999E+09,8.999999E+09,8.999999E+09]];
	LOCAL CONST Robtarget Tr_meulage_motif_1_P111 :=[[28.7191328125,147.822140625,74.1451640625],[0.0144291641931026,-0.0124615274841837,0.653500364086891,-0.756686053586129],[0,0,0,0],[8.999999E+09,8.999999E+09,8.999999E+09,8.999999E+09,8.999999E+09,8.999999E+09]];
	LOCAL CONST Robtarget Tr_meulage_motif_1_P112 :=[[29.678966796875,147.5419375,74.159328125],[0.0144291641931026,-0.0124615274841837,0.653500364086891,-0.756686053586129],[0,0,0,0],[8.999999E+09,8.999999E+09,8.999999E+09,8.999999E+09,8.999999E+09,8.999999E+09]];
	LOCAL CONST Robtarget Tr_meulage_motif_1_P113 :=[[30.63880078125,147.26171875,74.1734921875],[0.0144291641931026,-0.0124615274841837,0.653500364086891,-0.756686053586129],[0,0,0,0],[8.999999E+09,8.999999E+09,8.999999E+09,8.999999E+09,8.999999E+09,8.999999E+09]];
	LOCAL CONST Robtarget Tr_meulage_motif_1_P114 :=[[31.598634765625,146.981515625,74.18765625],[0.0144291641931026,-0.0124615274841837,0.653500364086891,-0.756686053586129],[0,0,0,0],[8.999999E+09,8.999999E+09,8.999999E+09,8.999999E+09,8.999999E+09,8.999999E+09]];
	LOCAL CONST Robtarget Tr_meulage_motif_1_P115 :=[[32.55846875,146.701296875,74.201828125],[0.0144291641931026,-0.0124615274841837,0.653500364086891,-0.756686053586129],[0,0,0,0],[8.999999E+09,8.999999E+09,8.999999E+09,8.999999E+09,8.999999E+09,8.999999E+09]];
	LOCAL CONST Robtarget Tr_meulage_motif_1_degg1 :=[[32.1812901878535,156.587592916837,72.7461884355788],[0.0144291641931026,-0.0124615274841837,0.653500364086891,-0.756686053586129],[0,0,0,0],[8.999999E+09,8.999999E+09,8.999999E+09,8.999999E+09,8.999999E+09,8.999999E+09]];
	LOCAL CONST Robtarget Tr_meulage_motif_1_degg2 :=[[25.0148975070704,344.427217711737,45.0890343365753],[0.0144291641931026,-0.0124615274841837,0.653500364086891,-0.756686053586129],[0,0,0,0],[8.999999E+09,8.999999E+09,8.999999E+09,8.999999E+09,8.999999E+09,8.999999E+09]];
	LOCAL CONST Robtarget Tr_meulage_motif_2_App1 :=[[305.400994088075,-35.870258705114,72.333920863134],[0.489692921812557,-0.497861576141384,-0.510298817976881,0.501926099839504],[0,0,0,0],[8.999999E+09,8.999999E+09,8.999999E+09,8.999999E+09,8.999999E+09,8.999999E+09]];
	LOCAL CONST Robtarget Tr_meulage_motif_2_App2 :=[[115.484807516904,-40.5568008258807,69.1909284650317],[0.489692921812557,-0.497861576141384,-0.510298817976881,0.501926099839504],[0,0,0,0],[8.999999E+09,8.999999E+09,8.999999E+09,8.999999E+09,8.999999E+09,8.999999E+09]];
	LOCAL CONST Robtarget Tr_meulage_motif_2_P0 :=[[105.48921875,-40.8034609375,69.0255078125],[0.489692921812557,-0.497861576141384,-0.510298817976881,0.501926099839504],[0,0,0,0],[8.999999E+09,8.999999E+09,8.999999E+09,8.999999E+09,8.999999E+09,8.999999E+09]];
	LOCAL CONST Robtarget Tr_meulage_motif_2_P1 :=[[105.4443046875,-39.80447265625,69.0257109375],[0.489692921812557,-0.497861576141384,-0.510298817976881,0.501926099839504],[0,0,0,0],[8.999999E+09,8.999999E+09,8.999999E+09,8.999999E+09,8.999999E+09,8.999999E+09]];
	LOCAL CONST Robtarget Tr_meulage_motif_2_P2 :=[[105.3993984375,-38.80548046875,69.02590625],[0.489692921812557,-0.497861576141384,-0.510298817976881,0.501926099839504],[0,0,0,0],[8.999999E+09,8.999999E+09,8.999999E+09,8.999999E+09,8.999999E+09,8.999999E+09]];
	LOCAL CONST Robtarget Tr_meulage_motif_2_P3 :=[[105.3544921875,-37.80648828125,69.026109375],[0.489692921812557,-0.497861576141384,-0.510298817976881,0.501926099839504],[0,0,0,0],[8.999999E+09,8.999999E+09,8.999999E+09,8.999999E+09,8.999999E+09,8.999999E+09]];
	LOCAL CONST Robtarget Tr_meulage_motif_2_P4 :=[[105.3095859375,-36.8075,69.0263125],[0.489692921812557,-0.497861576141384,-0.510298817976881,0.501926099839504],[0,0,0,0],[8.999999E+09,8.999999E+09,8.999999E+09,8.999999E+09,8.999999E+09,8.999999E+09]];
	LOCAL CONST Robtarget Tr_meulage_motif_2_P5 :=[[105.264671875,-35.8085078125,69.026515625],[0.489692921812557,-0.497861576141384,-0.510298817976881,0.501926099839504],[0,0,0,0],[8.999999E+09,8.999999E+09,8.999999E+09,8.999999E+09,8.999999E+09,8.999999E+09]];
	LOCAL CONST Robtarget Tr_meulage_motif_2_P6 :=[[105.219765625,-34.809515625,69.02671875],[0.489692921812557,-0.497861576141384,-0.510298817976881,0.501926099839504],[0,0,0,0],[8.999999E+09,8.999999E+09,8.999999E+09,8.999999E+09,8.999999E+09,8.999999E+09]];
	LOCAL CONST Robtarget Tr_meulage_motif_2_P7 :=[[105.174859375,-33.8105234375,69.026921875],[0.489692921812557,-0.497861576141384,-0.510298817976881,0.501926099839504],[0,0,0,0],[8.999999E+09,8.999999E+09,8.999999E+09,8.999999E+09,8.999999E+09,8.999999E+09]];
	LOCAL CONST Robtarget Tr_meulage_motif_2_P8 :=[[105.129953125,-32.81153515625,69.0271171875],[0.489692921812557,-0.497861576141384,-0.510298817976881,0.501926099839504],[0,0,0,0],[8.999999E+09,8.999999E+09,8.999999E+09,8.999999E+09,8.999999E+09,8.999999E+09]];
	LOCAL CONST Robtarget Tr_meulage_motif_2_P9 :=[[105.0850390625,-31.81254296875,69.0273203125],[0.489692921812557,-0.497861576141384,-0.510298817976881,0.501926099839504],[0,0,0,0],[8.999999E+09,8.999999E+09,8.999999E+09,8.999999E+09,8.999999E+09,8.999999E+09]];
	LOCAL CONST Robtarget Tr_meulage_motif_2_P10 :=[[105.0401328125,-30.81355078125,69.0275234375],[0.489692921812557,-0.497861576141384,-0.510298817976881,0.501926099839504],[0,0,0,0],[8.999999E+09,8.999999E+09,8.999999E+09,8.999999E+09,8.999999E+09,8.999999E+09]];
	LOCAL CONST Robtarget Tr_meulage_motif_2_P11 :=[[104.9952265625,-29.814560546875,69.0277265625],[0.489692921812557,-0.497861576141384,-0.510298817976881,0.501926099839504],[0,0,0,0],[8.999999E+09,8.999999E+09,8.999999E+09,8.999999E+09,8.999999E+09,8.999999E+09]];
	LOCAL CONST Robtarget Tr_meulage_motif_2_P12 :=[[104.9503203125,-28.815568359375,69.0279296875],[0.489692921812557,-0.497861576141384,-0.510298817976881,0.501926099839504],[0,0,0,0],[8.999999E+09,8.999999E+09,8.999999E+09,8.999999E+09,8.999999E+09,8.999999E+09]];
	LOCAL CONST Robtarget Tr_meulage_motif_2_P13 :=[[104.90540625,-27.816578125,69.028125],[0.489692921812557,-0.497861576141384,-0.510298817976881,0.501926099839504],[0,0,0,0],[8.999999E+09,8.999999E+09,8.999999E+09,8.999999E+09,8.999999E+09,8.999999E+09]];
	LOCAL CONST Robtarget Tr_meulage_motif_2_P14 :=[[104.8605,-26.817587890625,69.028328125],[0.489692921812557,-0.497861576141384,-0.510298817976881,0.501926099839504],[0,0,0,0],[8.999999E+09,8.999999E+09,8.999999E+09,8.999999E+09,8.999999E+09,8.999999E+09]];
	LOCAL CONST Robtarget Tr_meulage_motif_2_P15 :=[[104.81559375,-25.818595703125,69.02853125],[0.489692921812557,-0.497861576141384,-0.510298817976881,0.501926099839504],[0,0,0,0],[8.999999E+09,8.999999E+09,8.999999E+09,8.999999E+09,8.999999E+09,8.999999E+09]];
	LOCAL CONST Robtarget Tr_meulage_motif_2_P16 :=[[104.7706875,-24.81960546875,69.028734375],[0.489692921812557,-0.497861576141384,-0.510298817976881,0.501926099839504],[0,0,0,0],[8.999999E+09,8.999999E+09,8.999999E+09,8.999999E+09,8.999999E+09,8.999999E+09]];
	LOCAL CONST Robtarget Tr_meulage_motif_2_P17 :=[[104.7257734375,-23.82061328125,69.0289375],[0.489692921812557,-0.497861576141384,-0.510298817976881,0.501926099839504],[0,0,0,0],[8.999999E+09,8.999999E+09,8.999999E+09,8.999999E+09,8.999999E+09,8.999999E+09]];
	LOCAL CONST Robtarget Tr_meulage_motif_2_P18 :=[[104.6808671875,-22.821623046875,69.029140625],[0.489692921812557,-0.497861576141384,-0.510298817976881,0.501926099839504],[0,0,0,0],[8.999999E+09,8.999999E+09,8.999999E+09,8.999999E+09,8.999999E+09,8.999999E+09]];
	LOCAL CONST Robtarget Tr_meulage_motif_2_P19 :=[[104.637984375,-21.829962890625,68.9187578125],[0.489692921812557,-0.497861576141384,-0.510298817976881,0.501926099839504],[0,0,0,0],[8.999999E+09,8.999999E+09,8.999999E+09,8.999999E+09,8.999999E+09,8.999999E+09]];
	LOCAL CONST Robtarget Tr_meulage_motif_2_P20 :=[[104.5987109375,-20.88423046875,68.70778125],[0.489692921812557,-0.497861576141384,-0.510298817976881,0.501926099839504],[0,0,0,0],[8.999999E+09,8.999999E+09,8.999999E+09,8.999999E+09,8.999999E+09,8.999999E+09]];
	LOCAL CONST Robtarget Tr_meulage_motif_2_P21 :=[[104.5645703125,-20.032130859375,68.4361484375],[0.489692921812557,-0.497861576141384,-0.510298817976881,0.501926099839504],[0,0,0,0],[8.999999E+09,8.999999E+09,8.999999E+09,8.999999E+09,8.999999E+09,8.999999E+09]];
	LOCAL CONST Robtarget Tr_meulage_motif_2_P22 :=[[104.5351171875,-19.282703125,68.160390625],[0.489692921812557,-0.497861576141384,-0.510298817976881,0.501926099839504],[0,0,0,0],[8.999999E+09,8.999999E+09,8.999999E+09,8.999999E+09,8.999999E+09,8.999999E+09]];
	LOCAL CONST Robtarget Tr_meulage_motif_2_P23 :=[[104.49509375,-18.182205078125,67.5445625],[0.489692921812557,-0.497861576141384,-0.510298817976881,0.501926099839504],[0,0,0,0],[8.999999E+09,8.999999E+09,8.999999E+09,8.999999E+09,8.999999E+09,8.999999E+09]];
	LOCAL CONST Robtarget Tr_meulage_motif_2_P24 :=[[104.4620703125,-17.158607421875,66.6972109375],[0.489692921812557,-0.497861576141384,-0.510298817976881,0.501926099839504],[0,0,0,0],[8.999999E+09,8.999999E+09,8.999999E+09,8.999999E+09,8.999999E+09,8.999999E+09]];
	LOCAL CONST Robtarget Tr_meulage_motif_2_P25 :=[[104.4396640625,-16.310896484375,65.673625],[0.489692921812557,-0.497861576141384,-0.510298817976881,0.501926099839504],[0,0,0,0],[8.999999E+09,8.999999E+09,8.999999E+09,8.999999E+09,8.999999E+09,8.999999E+09]];
	LOCAL CONST Robtarget Tr_meulage_motif_2_P26 :=[[104.4348125,-15.822240234375,64.55766796875],[0.489692921812557,-0.497861576141384,-0.510298817976881,0.501926099839504],[0,0,0,0],[8.999999E+09,8.999999E+09,8.999999E+09,8.999999E+09,8.999999E+09,8.999999E+09]];
	LOCAL CONST Robtarget Tr_meulage_motif_2_P27 :=[[104.4442421875,-15.7945859375,63.86178515625],[0.489692921812557,-0.497861576141384,-0.510298817976881,0.501926099839504],[0,0,0,0],[8.999999E+09,8.999999E+09,8.999999E+09,8.999999E+09,8.999999E+09,8.999999E+09]];
	LOCAL CONST Robtarget Tr_meulage_motif_2_P28 :=[[104.4543515625,-15.793998046875,63.20061328125],[0.489692921812557,-0.497861576141384,-0.510298817976881,0.501926099839504],[0,0,0,0],[8.999999E+09,8.999999E+09,8.999999E+09,8.999999E+09,8.999999E+09,8.999999E+09]];
	LOCAL CONST Robtarget Tr_meulage_motif_2_P29 :=[[104.466921875,-15.8482294921875,62.5395859375],[0.489692921812557,-0.497861576141384,-0.510298817976881,0.501926099839504],[0,0,0,0],[8.999999E+09,8.999999E+09,8.999999E+09,8.999999E+09,8.999999E+09,8.999999E+09]];
	LOCAL CONST Robtarget Tr_meulage_motif_2_P30 :=[[104.5061484375,-16.3449658203125,61.4378671875],[0.489692921812557,-0.497861576141384,-0.510298817976881,0.501926099839504],[0,0,0,0],[8.999999E+09,8.999999E+09,8.999999E+09,8.999999E+09,8.999999E+09,8.999999E+09]];
	LOCAL CONST Robtarget Tr_meulage_motif_2_P31 :=[[104.5600078125,-17.19983203125,60.4311875],[0.489692921812557,-0.497861576141384,-0.510298817976881,0.501926099839504],[0,0,0,0],[8.999999E+09,8.999999E+09,8.999999E+09,8.999999E+09,8.999999E+09,8.999999E+09]];
	LOCAL CONST Robtarget Tr_meulage_motif_2_P32 :=[[104.6186484375,-18.22146875,59.602203125],[0.489692921812557,-0.497861576141384,-0.510298817976881,0.501926099839504],[0,0,0,0],[8.999999E+09,8.999999E+09,8.999999E+09,8.999999E+09,8.999999E+09,8.999999E+09]];
	LOCAL CONST Robtarget Tr_meulage_motif_2_P33 :=[[104.6555546875,-18.907517578125,59.206359375],[0.489692921812557,-0.497861576141384,-0.510298817976881,0.501926099839504],[0,0,0,0],[8.999999E+09,8.999999E+09,8.999999E+09,8.999999E+09,8.999999E+09,8.999999E+09]];
	LOCAL CONST Robtarget Tr_meulage_motif_2_P34 :=[[104.7150234375,-20.0640703125,58.71865234375],[0.489692921812557,-0.497861576141384,-0.510298817976881,0.501926099839504],[0,0,0,0],[8.999999E+09,8.999999E+09,8.999999E+09,8.999999E+09,8.999999E+09,8.999999E+09]];
	LOCAL CONST Robtarget Tr_meulage_motif_2_P35 :=[[104.7570078125,-20.908015625,58.45441796875],[0.489692921812557,-0.497861576141384,-0.510298817976881,0.501926099839504],[0,0,0,0],[8.999999E+09,8.999999E+09,8.999999E+09,8.999999E+09,8.999999E+09,8.999999E+09]];
	LOCAL CONST Robtarget Tr_meulage_motif_2_P36 :=[[104.8019921875,-21.838892578125,58.24978515625],[0.489692921812557,-0.497861576141384,-0.510298817976881,0.501926099839504],[0,0,0,0],[8.999999E+09,8.999999E+09,8.999999E+09,8.999999E+09,8.999999E+09,8.999999E+09]];
	LOCAL CONST Robtarget Tr_meulage_motif_2_P37 :=[[104.8477265625,-22.819369140625,58.1410078125],[0.489692921812557,-0.497861576141384,-0.510298817976881,0.501926099839504],[0,0,0,0],[8.999999E+09,8.999999E+09,8.999999E+09,8.999999E+09,8.999999E+09,8.999999E+09]];
	LOCAL CONST Robtarget Tr_meulage_motif_2_P38 :=[[104.8939921875,-23.810830078125,58.0302265625],[0.489692921812557,-0.497861576141384,-0.510298817976881,0.501926099839504],[0,0,0,0],[8.999999E+09,8.999999E+09,8.999999E+09,8.999999E+09,8.999999E+09,8.999999E+09]];
	LOCAL CONST Robtarget Tr_meulage_motif_2_P39 :=[[104.93890625,-24.809822265625,58.0300234375],[0.489692921812557,-0.497861576141384,-0.510298817976881,0.501926099839504],[0,0,0,0],[8.999999E+09,8.999999E+09,8.999999E+09,8.999999E+09,8.999999E+09,8.999999E+09]];
	LOCAL CONST Robtarget Tr_meulage_motif_2_P40 :=[[104.9838125,-25.8088125,58.02982421875],[0.489692921812557,-0.497861576141384,-0.510298817976881,0.501926099839504],[0,0,0,0],[8.999999E+09,8.999999E+09,8.999999E+09,8.999999E+09,8.999999E+09,8.999999E+09]];
	LOCAL CONST Robtarget Tr_meulage_motif_2_P41 :=[[105.02871875,-26.8078046875,58.02962109375],[0.489692921812557,-0.497861576141384,-0.510298817976881,0.501926099839504],[0,0,0,0],[8.999999E+09,8.999999E+09,8.999999E+09,8.999999E+09,8.999999E+09,8.999999E+09]];
	LOCAL CONST Robtarget Tr_meulage_motif_2_P42 :=[[105.073625,-27.806794921875,58.02941796875],[0.489692921812557,-0.497861576141384,-0.510298817976881,0.501926099839504],[0,0,0,0],[8.999999E+09,8.999999E+09,8.999999E+09,8.999999E+09,8.999999E+09,8.999999E+09]];
	LOCAL CONST Robtarget Tr_meulage_motif_2_P43 :=[[105.1185390625,-28.805787109375,58.02921875],[0.489692921812557,-0.497861576141384,-0.510298817976881,0.501926099839504],[0,0,0,0],[8.999999E+09,8.999999E+09,8.999999E+09,8.999999E+09,8.999999E+09,8.999999E+09]];
	LOCAL CONST Robtarget Tr_meulage_motif_2_P44 :=[[105.1634453125,-29.80477734375,58.029015625],[0.489692921812557,-0.497861576141384,-0.510298817976881,0.501926099839504],[0,0,0,0],[8.999999E+09,8.999999E+09,8.999999E+09,8.999999E+09,8.999999E+09,8.999999E+09]];
	LOCAL CONST Robtarget Tr_meulage_motif_2_P45 :=[[105.2083515625,-30.80376953125,58.0288125],[0.489692921812557,-0.497861576141384,-0.510298817976881,0.501926099839504],[0,0,0,0],[8.999999E+09,8.999999E+09,8.999999E+09,8.999999E+09,8.999999E+09,8.999999E+09]];
	LOCAL CONST Robtarget Tr_meulage_motif_2_P46 :=[[105.2532578125,-31.802759765625,58.02861328125],[0.489692921812557,-0.497861576141384,-0.510298817976881,0.501926099839504],[0,0,0,0],[8.999999E+09,8.999999E+09,8.999999E+09,8.999999E+09,8.999999E+09,8.999999E+09]];
	LOCAL CONST Robtarget Tr_meulage_motif_2_P47 :=[[105.2981640625,-32.80175,58.02841015625],[0.489692921812557,-0.497861576141384,-0.510298817976881,0.501926099839504],[0,0,0,0],[8.999999E+09,8.999999E+09,8.999999E+09,8.999999E+09,8.999999E+09,8.999999E+09]];
	LOCAL CONST Robtarget Tr_meulage_motif_2_P48 :=[[105.343078125,-33.8007421875,58.0282109375],[0.489692921812557,-0.497861576141384,-0.510298817976881,0.501926099839504],[0,0,0,0],[8.999999E+09,8.999999E+09,8.999999E+09,8.999999E+09,8.999999E+09,8.999999E+09]];
	LOCAL CONST Robtarget Tr_meulage_motif_2_P49 :=[[105.38934375,-34.792203125,57.9174296875],[0.489692921812557,-0.497861576141384,-0.510298817976881,0.501926099839504],[0,0,0,0],[8.999999E+09,8.999999E+09,8.999999E+09,8.999999E+09,8.999999E+09,8.999999E+09]];
	LOCAL CONST Robtarget Tr_meulage_motif_2_P50 :=[[105.435078125,-35.7375625,57.70607421875],[0.489692921812557,-0.497861576141384,-0.510298817976881,0.501926099839504],[0,0,0,0],[8.999999E+09,8.999999E+09,8.999999E+09,8.999999E+09,8.999999E+09,8.999999E+09]];
	LOCAL CONST Robtarget Tr_meulage_motif_2_P51 :=[[105.4775234375,-36.5891796875,57.43408984375],[0.489692921812557,-0.497861576141384,-0.510298817976881,0.501926099839504],[0,0,0,0],[8.999999E+09,8.999999E+09,8.999999E+09,8.999999E+09,8.999999E+09,8.999999E+09]];
	LOCAL CONST Robtarget Tr_meulage_motif_2_P52 :=[[105.5141328125,-37.29969140625,57.129828125],[0.489692921812557,-0.497861576141384,-0.510298817976881,0.501926099839504],[0,0,0,0],[8.999999E+09,8.999999E+09,8.999999E+09,8.999999E+09,8.999999E+09,8.999999E+09]];
	LOCAL CONST Robtarget Tr_meulage_motif_2_P53 :=[[105.57071875,-38.33252734375,56.4671640625],[0.489692921812557,-0.497861576141384,-0.510298817976881,0.501926099839504],[0,0,0,0],[8.999999E+09,8.999999E+09,8.999999E+09,8.999999E+09,8.999999E+09,8.999999E+09]];
	LOCAL CONST Robtarget Tr_meulage_motif_2_P54 :=[[105.625015625,-39.23275,55.56515234375],[0.489692921812557,-0.497861576141384,-0.510298817976881,0.501926099839504],[0,0,0,0],[8.999999E+09,8.999999E+09,8.999999E+09,8.999999E+09,8.999999E+09,8.999999E+09]];
	LOCAL CONST Robtarget Tr_meulage_motif_2_P55 :=[[105.6650390625,-39.76625,54.5191328125],[0.489692921812557,-0.497861576141384,-0.510298817976881,0.501926099839504],[0,0,0,0],[8.999999E+09,8.999999E+09,8.999999E+09,8.999999E+09,8.999999E+09,8.999999E+09]];
	LOCAL CONST Robtarget Tr_meulage_motif_2_P56 :=[[105.6839375,-39.95023046875,53.8259609375],[0.489692921812557,-0.497861576141384,-0.510298817976881,0.501926099839504],[0,0,0,0],[8.999999E+09,8.999999E+09,8.999999E+09,8.999999E+09,8.999999E+09,8.999999E+09]];
	LOCAL CONST Robtarget Tr_meulage_motif_2_P57 :=[[105.698578125,-40.01332421875,53.0560390625],[0.489692921812557,-0.497861576141384,-0.510298817976881,0.501926099839504],[0,0,0,0],[8.999999E+09,8.999999E+09,8.999999E+09,8.999999E+09,8.999999E+09,8.999999E+09]];
	LOCAL CONST Robtarget Tr_meulage_motif_2_P58 :=[[105.70734375,-39.94576953125,52.286265625],[0.489692921812557,-0.497861576141384,-0.510298817976881,0.501926099839504],[0,0,0,0],[8.999999E+09,8.999999E+09,8.999999E+09,8.999999E+09,8.999999E+09,8.999999E+09]];
	LOCAL CONST Robtarget Tr_meulage_motif_2_P59 :=[[105.705453125,-39.52561328125,51.17823046875],[0.489692921812557,-0.497861576141384,-0.510298817976881,0.501926099839504],[0,0,0,0],[8.999999E+09,8.999999E+09,8.999999E+09,8.999999E+09,8.999999E+09,8.999999E+09]];
	LOCAL CONST Robtarget Tr_meulage_motif_2_P60 :=[[105.695796875,-39.1111953125,50.5926953125],[0.489692921812557,-0.497861576141384,-0.510298817976881,0.501926099839504],[0,0,0,0],[8.999999E+09,8.999999E+09,8.999999E+09,8.999999E+09,8.999999E+09,8.999999E+09]];
	LOCAL CONST Robtarget Tr_meulage_motif_2_P61 :=[[105.66953125,-38.2241796875,49.7058515625],[0.489692921812557,-0.497861576141384,-0.510298817976881,0.501926099839504],[0,0,0,0],[8.999999E+09,8.999999E+09,8.999999E+09,8.999999E+09,8.999999E+09,8.999999E+09]];
	LOCAL CONST Robtarget Tr_meulage_motif_2_P62 :=[[105.6495625,-37.63871484375,49.29170703125],[0.489692921812557,-0.497861576141384,-0.510298817976881,0.501926099839504],[0,0,0,0],[8.999999E+09,8.999999E+09,8.999999E+09,8.999999E+09,8.999999E+09,8.999999E+09]];
	LOCAL CONST Robtarget Tr_meulage_motif_2_P63 :=[[105.6076796875,-36.52144921875,48.74790234375],[0.489692921812557,-0.497861576141384,-0.510298817976881,0.501926099839504],[0,0,0,0],[8.999999E+09,8.999999E+09,8.999999E+09,8.999999E+09,8.999999E+09,8.999999E+09]];
	LOCAL CONST Robtarget Tr_meulage_motif_2_P64 :=[[105.575125,-35.69642578125,48.45260546875],[0.489692921812557,-0.497861576141384,-0.510298817976881,0.501926099839504],[0,0,0,0],[8.999999E+09,8.999999E+09,8.999999E+09,8.999999E+09,8.999999E+09,8.999999E+09]];
	LOCAL CONST Robtarget Tr_meulage_motif_2_P65 :=[[105.5363984375,-34.7651875,48.24834765625],[0.489692921812557,-0.497861576141384,-0.510298817976881,0.501926099839504],[0,0,0,0],[8.999999E+09,8.999999E+09,8.999999E+09,8.999999E+09,8.999999E+09,8.999999E+09]];
	LOCAL CONST Robtarget Tr_meulage_motif_2_P66 :=[[105.4939765625,-33.784515625,48.13996484375],[0.489692921812557,-0.497861576141384,-0.510298817976881,0.501926099839504],[0,0,0,0],[8.999999E+09,8.999999E+09,8.999999E+09,8.999999E+09,8.999999E+09,8.999999E+09]];
	LOCAL CONST Robtarget Tr_meulage_motif_2_P67 :=[[105.45109375,-32.79285546875,48.0295859375],[0.489692921812557,-0.497861576141384,-0.510298817976881,0.501926099839504],[0,0,0,0],[8.999999E+09,8.999999E+09,8.999999E+09,8.999999E+09,8.999999E+09,8.999999E+09]];
	LOCAL CONST Robtarget Tr_meulage_motif_2_P68 :=[[105.4061875,-31.7938671875,48.02978515625],[0.489692921812557,-0.497861576141384,-0.510298817976881,0.501926099839504],[0,0,0,0],[8.999999E+09,8.999999E+09,8.999999E+09,8.999999E+09,8.999999E+09,8.999999E+09]];
	LOCAL CONST Robtarget Tr_meulage_motif_2_P69 :=[[105.3612734375,-30.794875,48.02998828125],[0.489692921812557,-0.497861576141384,-0.510298817976881,0.501926099839504],[0,0,0,0],[8.999999E+09,8.999999E+09,8.999999E+09,8.999999E+09,8.999999E+09,8.999999E+09]];
	LOCAL CONST Robtarget Tr_meulage_motif_2_P70 :=[[105.3163671875,-29.795884765625,48.0301875],[0.489692921812557,-0.497861576141384,-0.510298817976881,0.501926099839504],[0,0,0,0],[8.999999E+09,8.999999E+09,8.999999E+09,8.999999E+09,8.999999E+09,8.999999E+09]];
	LOCAL CONST Robtarget Tr_meulage_motif_2_P71 :=[[105.2714609375,-28.796892578125,48.030390625],[0.489692921812557,-0.497861576141384,-0.510298817976881,0.501926099839504],[0,0,0,0],[8.999999E+09,8.999999E+09,8.999999E+09,8.999999E+09,8.999999E+09,8.999999E+09]];
	LOCAL CONST Robtarget Tr_meulage_motif_2_P72 :=[[105.2265546875,-27.79790234375,48.03059375],[0.489692921812557,-0.497861576141384,-0.510298817976881,0.501926099839504],[0,0,0,0],[8.999999E+09,8.999999E+09,8.999999E+09,8.999999E+09,8.999999E+09,8.999999E+09]];
	LOCAL CONST Robtarget Tr_meulage_motif_2_P73 :=[[105.181640625,-26.79891015625,48.03079296875],[0.489692921812557,-0.497861576141384,-0.510298817976881,0.501926099839504],[0,0,0,0],[8.999999E+09,8.999999E+09,8.999999E+09,8.999999E+09,8.999999E+09,8.999999E+09]];
	LOCAL CONST Robtarget Tr_meulage_motif_2_P74 :=[[105.136734375,-25.799919921875,48.03099609375],[0.489692921812557,-0.497861576141384,-0.510298817976881,0.501926099839504],[0,0,0,0],[8.999999E+09,8.999999E+09,8.999999E+09,8.999999E+09,8.999999E+09,8.999999E+09]];
	LOCAL CONST Robtarget Tr_meulage_motif_2_P75 :=[[105.091828125,-24.800927734375,48.03119921875],[0.489692921812557,-0.497861576141384,-0.510298817976881,0.501926099839504],[0,0,0,0],[8.999999E+09,8.999999E+09,8.999999E+09,8.999999E+09,8.999999E+09,8.999999E+09]];
	LOCAL CONST Robtarget Tr_meulage_motif_2_P76 :=[[105.046921875,-23.8019375,48.0313984375],[0.489692921812557,-0.497861576141384,-0.510298817976881,0.501926099839504],[0,0,0,0],[8.999999E+09,8.999999E+09,8.999999E+09,8.999999E+09,8.999999E+09,8.999999E+09]];
	LOCAL CONST Robtarget Tr_meulage_motif_2_P77 :=[[105.0020078125,-22.802947265625,48.0316015625],[0.489692921812557,-0.497861576141384,-0.510298817976881,0.501926099839504],[0,0,0,0],[8.999999E+09,8.999999E+09,8.999999E+09,8.999999E+09,8.999999E+09,8.999999E+09]];
	LOCAL CONST Robtarget Tr_meulage_motif_2_P78 :=[[104.959125,-21.811287109375,47.92122265625],[0.489692921812557,-0.497861576141384,-0.510298817976881,0.501926099839504],[0,0,0,0],[8.999999E+09,8.999999E+09,8.999999E+09,8.999999E+09,8.999999E+09,8.999999E+09]];
	LOCAL CONST Robtarget Tr_meulage_motif_2_P79 :=[[104.9198515625,-20.8655546875,47.71025],[0.489692921812557,-0.497861576141384,-0.510298817976881,0.501926099839504],[0,0,0,0],[8.999999E+09,8.999999E+09,8.999999E+09,8.999999E+09,8.999999E+09,8.999999E+09]];
	LOCAL CONST Robtarget Tr_meulage_motif_2_P80 :=[[104.88571875,-20.013453125,47.438609375],[0.489692921812557,-0.497861576141384,-0.510298817976881,0.501926099839504],[0,0,0,0],[8.999999E+09,8.999999E+09,8.999999E+09,8.999999E+09,8.999999E+09,8.999999E+09]];
	LOCAL CONST Robtarget Tr_meulage_motif_2_P81 :=[[104.8562578125,-19.26402734375,47.16285546875],[0.489692921812557,-0.497861576141384,-0.510298817976881,0.501926099839504],[0,0,0,0],[8.999999E+09,8.999999E+09,8.999999E+09,8.999999E+09,8.999999E+09,8.999999E+09]];
	LOCAL CONST Robtarget Tr_meulage_motif_2_P82 :=[[104.816234375,-18.16352734375,46.5470234375],[0.489692921812557,-0.497861576141384,-0.510298817976881,0.501926099839504],[0,0,0,0],[8.999999E+09,8.999999E+09,8.999999E+09,8.999999E+09,8.999999E+09,8.999999E+09]];
	LOCAL CONST Robtarget Tr_meulage_motif_2_P83 :=[[104.7869375,-17.206978515625,45.65335546875],[0.489692921812557,-0.497861576141384,-0.510298817976881,0.501926099839504],[0,0,0,0],[8.999999E+09,8.999999E+09,8.999999E+09,8.999999E+09,8.999999E+09,8.999999E+09]];
	LOCAL CONST Robtarget Tr_meulage_motif_2_P84 :=[[104.7761953125,-16.59750390625,44.56760546875],[0.489692921812557,-0.497861576141384,-0.510298817976881,0.501926099839504],[0,0,0,0],[8.999999E+09,8.999999E+09,8.999999E+09,8.999999E+09,8.999999E+09,8.999999E+09]];
	LOCAL CONST Robtarget Tr_meulage_motif_2_P85 :=[[104.783640625,-16.427486328125,43.58337890625],[0.489692921812557,-0.497861576141384,-0.510298817976881,0.501926099839504],[0,0,0,0],[8.999999E+09,8.999999E+09,8.999999E+09,8.999999E+09,8.999999E+09,8.999999E+09]];
	LOCAL CONST Robtarget Tr_meulage_motif_2_P86 :=[[104.7926796875,-16.558640625,43.37871875],[0.489692921812557,-0.497861576141384,-0.510298817976881,0.501926099839504],[0,0,0,0],[8.999999E+09,8.999999E+09,8.999999E+09,8.999999E+09,8.999999E+09,8.999999E+09]];
	LOCAL CONST Robtarget Tr_meulage_motif_2_P87 :=[[104.809328125,-16.681244140625,42.652375],[0.489692921812557,-0.497861576141384,-0.510298817976881,0.501926099839504],[0,0,0,0],[8.999999E+09,8.999999E+09,8.999999E+09,8.999999E+09,8.999999E+09,8.999999E+09]];
	LOCAL CONST Robtarget Tr_meulage_motif_2_P88 :=[[104.8543671875,-17.363720703125,41.71544140625],[0.489692921812557,-0.497861576141384,-0.510298817976881,0.501926099839504],[0,0,0,0],[8.999999E+09,8.999999E+09,8.999999E+09,8.999999E+09,8.999999E+09,8.999999E+09]];
	LOCAL CONST Robtarget Tr_meulage_motif_2_P89 :=[[104.8865078125,-17.92037109375,41.2515703125],[0.489692921812557,-0.497861576141384,-0.510298817976881,0.501926099839504],[0,0,0,0],[8.999999E+09,8.999999E+09,8.999999E+09,8.999999E+09,8.999999E+09,8.999999E+09]];
	LOCAL CONST Robtarget Tr_meulage_motif_2_P90 :=[[104.945375,-19.049072265625,40.72096484375],[0.489692921812557,-0.497861576141384,-0.510298817976881,0.501926099839504],[0,0,0,0],[8.999999E+09,8.999999E+09,8.999999E+09,8.999999E+09,8.999999E+09,8.999999E+09]];
	LOCAL CONST Robtarget Tr_meulage_motif_2_P91 :=[[104.9873671875,-19.893015625,40.456734375],[0.489692921812557,-0.497861576141384,-0.510298817976881,0.501926099839504],[0,0,0,0],[8.999999E+09,8.999999E+09,8.999999E+09,8.999999E+09,8.999999E+09,8.999999E+09]];
	LOCAL CONST Robtarget Tr_meulage_motif_2_P92 :=[[105.03234375,-20.823892578125,40.2521015625],[0.489692921812557,-0.497861576141384,-0.510298817976881,0.501926099839504],[0,0,0,0],[8.999999E+09,8.999999E+09,8.999999E+09,8.999999E+09,8.999999E+09,8.999999E+09]];
	LOCAL CONST Robtarget Tr_meulage_motif_2_P93 :=[[105.0780859375,-21.804369140625,40.1433203125],[0.489692921812557,-0.497861576141384,-0.510298817976881,0.501926099839504],[0,0,0,0],[8.999999E+09,8.999999E+09,8.999999E+09,8.999999E+09,8.999999E+09,8.999999E+09]];
	LOCAL CONST Robtarget Tr_meulage_motif_2_P94 :=[[105.1243515625,-22.79583203125,40.0325390625],[0.489692921812557,-0.497861576141384,-0.510298817976881,0.501926099839504],[0,0,0,0],[8.999999E+09,8.999999E+09,8.999999E+09,8.999999E+09,8.999999E+09,8.999999E+09]];
	LOCAL CONST Robtarget Tr_meulage_motif_2_P95 :=[[105.1692578125,-23.794822265625,40.03233984375],[0.489692921812557,-0.497861576141384,-0.510298817976881,0.501926099839504],[0,0,0,0],[8.999999E+09,8.999999E+09,8.999999E+09,8.999999E+09,8.999999E+09,8.999999E+09]];
	LOCAL CONST Robtarget Tr_meulage_motif_2_P96 :=[[105.2141640625,-24.793814453125,40.03213671875],[0.489692921812557,-0.497861576141384,-0.510298817976881,0.501926099839504],[0,0,0,0],[8.999999E+09,8.999999E+09,8.999999E+09,8.999999E+09,8.999999E+09,8.999999E+09]];
	LOCAL CONST Robtarget Tr_meulage_motif_2_P97 :=[[105.259078125,-25.7928046875,40.03193359375],[0.489692921812557,-0.497861576141384,-0.510298817976881,0.501926099839504],[0,0,0,0],[8.999999E+09,8.999999E+09,8.999999E+09,8.999999E+09,8.999999E+09,8.999999E+09]];
	LOCAL CONST Robtarget Tr_meulage_motif_2_P98 :=[[105.303984375,-26.791796875,40.031734375],[0.489692921812557,-0.497861576141384,-0.510298817976881,0.501926099839504],[0,0,0,0],[8.999999E+09,8.999999E+09,8.999999E+09,8.999999E+09,8.999999E+09,8.999999E+09]];
	LOCAL CONST Robtarget Tr_meulage_motif_2_P99 :=[[105.348890625,-27.790787109375,40.03153125],[0.489692921812557,-0.497861576141384,-0.510298817976881,0.501926099839504],[0,0,0,0],[8.999999E+09,8.999999E+09,8.999999E+09,8.999999E+09,8.999999E+09,8.999999E+09]];
	LOCAL CONST Robtarget Tr_meulage_motif_2_P100 :=[[105.393796875,-28.78977734375,40.031328125],[0.489692921812557,-0.497861576141384,-0.510298817976881,0.501926099839504],[0,0,0,0],[8.999999E+09,8.999999E+09,8.999999E+09,8.999999E+09,8.999999E+09,8.999999E+09]];
	LOCAL CONST Robtarget Tr_meulage_motif_2_P101 :=[[105.4387109375,-29.78876953125,40.03112890625],[0.489692921812557,-0.497861576141384,-0.510298817976881,0.501926099839504],[0,0,0,0],[8.999999E+09,8.999999E+09,8.999999E+09,8.999999E+09,8.999999E+09,8.999999E+09]];
	LOCAL CONST Robtarget Tr_meulage_motif_2_P102 :=[[105.4836171875,-30.787759765625,40.03092578125],[0.489692921812557,-0.497861576141384,-0.510298817976881,0.501926099839504],[0,0,0,0],[8.999999E+09,8.999999E+09,8.999999E+09,8.999999E+09,8.999999E+09,8.999999E+09]];
	LOCAL CONST Robtarget Tr_meulage_motif_2_P103 :=[[105.5285234375,-31.786751953125,40.03072265625],[0.489692921812557,-0.497861576141384,-0.510298817976881,0.501926099839504],[0,0,0,0],[8.999999E+09,8.999999E+09,8.999999E+09,8.999999E+09,8.999999E+09,8.999999E+09]];
	LOCAL CONST Robtarget Tr_meulage_motif_2_P104 :=[[105.5734296875,-32.7857421875,40.0305234375],[0.489692921812557,-0.497861576141384,-0.510298817976881,0.501926099839504],[0,0,0,0],[8.999999E+09,8.999999E+09,8.999999E+09,8.999999E+09,8.999999E+09,8.999999E+09]];
	LOCAL CONST Robtarget Tr_meulage_motif_2_P105 :=[[105.61834375,-33.784734375,40.0303203125],[0.489692921812557,-0.497861576141384,-0.510298817976881,0.501926099839504],[0,0,0,0],[8.999999E+09,8.999999E+09,8.999999E+09,8.999999E+09,8.999999E+09,8.999999E+09]];
	LOCAL CONST Robtarget Tr_meulage_motif_2_P106 :=[[105.66325,-34.7837265625,40.03012109375],[0.489692921812557,-0.497861576141384,-0.510298817976881,0.501926099839504],[0,0,0,0],[8.999999E+09,8.999999E+09,8.999999E+09,8.999999E+09,8.999999E+09,8.999999E+09]];
	LOCAL CONST Robtarget Tr_meulage_motif_2_P107 :=[[105.70815625,-35.78271484375,40.02991796875],[0.489692921812557,-0.497861576141384,-0.510298817976881,0.501926099839504],[0,0,0,0],[8.999999E+09,8.999999E+09,8.999999E+09,8.999999E+09,8.999999E+09,8.999999E+09]];
	LOCAL CONST Robtarget Tr_meulage_motif_2_P108 :=[[105.7530625,-36.78170703125,40.02971484375],[0.489692921812557,-0.497861576141384,-0.510298817976881,0.501926099839504],[0,0,0,0],[8.999999E+09,8.999999E+09,8.999999E+09,8.999999E+09,8.999999E+09,8.999999E+09]];
	LOCAL CONST Robtarget Tr_meulage_motif_2_P109 :=[[105.7979765625,-37.78069921875,40.029515625],[0.489692921812557,-0.497861576141384,-0.510298817976881,0.501926099839504],[0,0,0,0],[8.999999E+09,8.999999E+09,8.999999E+09,8.999999E+09,8.999999E+09,8.999999E+09]];
	LOCAL CONST Robtarget Tr_meulage_motif_2_P110 :=[[105.8428828125,-38.7796875,40.0293125],[0.489692921812557,-0.497861576141384,-0.510298817976881,0.501926099839504],[0,0,0,0],[8.999999E+09,8.999999E+09,8.999999E+09,8.999999E+09,8.999999E+09,8.999999E+09]];
	LOCAL CONST Robtarget Tr_meulage_motif_2_P111 :=[[105.8877890625,-39.7786796875,40.029109375],[0.489692921812557,-0.497861576141384,-0.510298817976881,0.501926099839504],[0,0,0,0],[8.999999E+09,8.999999E+09,8.999999E+09,8.999999E+09,8.999999E+09,8.999999E+09]];
	LOCAL CONST Robtarget Tr_meulage_motif_2_P112 :=[[105.9326953125,-40.777671875,40.02891015625],[0.489692921812557,-0.497861576141384,-0.510298817976881,0.501926099839504],[0,0,0,0],[8.999999E+09,8.999999E+09,8.999999E+09,8.999999E+09,8.999999E+09,8.999999E+09]];
	LOCAL CONST Robtarget Tr_meulage_motif_2_P113 :=[[105.9776015625,-41.7766640625,40.02870703125],[0.489692921812557,-0.497861576141384,-0.510298817976881,0.501926099839504],[0,0,0,0],[8.999999E+09,8.999999E+09,8.999999E+09,8.999999E+09,8.999999E+09,8.999999E+09]];
	LOCAL CONST Robtarget Tr_meulage_motif_2_P114 :=[[106.022515625,-42.77565234375,40.02850390625],[0.489692921812557,-0.497861576141384,-0.510298817976881,0.501926099839504],[0,0,0,0],[8.999999E+09,8.999999E+09,8.999999E+09,8.999999E+09,8.999999E+09,8.999999E+09]];
	LOCAL CONST Robtarget Tr_meulage_motif_2_P115 :=[[106.067421875,-43.77464453125,40.0283046875],[0.489692921812557,-0.497861576141384,-0.510298817976881,0.501926099839504],[0,0,0,0],[8.999999E+09,8.999999E+09,8.999999E+09,8.999999E+09,8.999999E+09,8.999999E+09]];
	LOCAL CONST Robtarget Tr_meulage_motif_2_degg1 :=[[116.063010641904,-43.5279844196307,40.1937253400317],[0.489692921812557,-0.497861576141384,-0.510298817976881,0.501926099839504],[0,0,0,0],[8.999999E+09,8.999999E+09,8.999999E+09,8.999999E+09,8.999999E+09,8.999999E+09]];
	LOCAL CONST Robtarget Tr_meulage_motif_2_degg2 :=[[305.979197213074,-38.841442298864,43.336717738134],[0.489692921812557,-0.497861576141384,-0.510298817976881,0.501926099839504],[0,0,0,0],[8.999999E+09,8.999999E+09,8.999999E+09,8.999999E+09,8.999999E+09,8.999999E+09]];
	LOCAL CONST Robtarget Tr_meulage_bavure_App1 :=[[308.441236825011,-122.030351970132,111.383371409359],[0.489762976384074,-0.474720376740169,-0.508967406182428,0.525095201192142],[0,0,0,0],[8.999999E+09,8.999999E+09,8.999999E+09,8.999999E+09,8.999999E+09,8.999999E+09]];
	LOCAL CONST Robtarget Tr_meulage_bavure_App2 :=[[118.993459106876,-135.237585567257,117.308613882968],[0.489762976384074,-0.474720376740169,-0.508967406182428,0.525095201192142],[0,0,0,0],[8.999999E+09,8.999999E+09,8.999999E+09,8.999999E+09,8.999999E+09,8.999999E+09]];
	LOCAL CONST Robtarget Tr_meulage_bavure_P0 :=[[109.0225234375,-135.932703125,117.62046875],[0.489762976384074,-0.474720376740169,-0.508967406182428,0.525095201192142],[0,0,0,0],[8.999999E+09,8.999999E+09,8.999999E+09,8.999999E+09,8.999999E+09,8.999999E+09]];
	LOCAL CONST Robtarget Tr_meulage_bavure_P1 :=[[108.9333828125,-135.5015,117.5613984375],[0.49011118687594,-0.475004937192246,-0.508647109674635,0.52482325783228],[0,0,0,0],[8.999999E+09,8.999999E+09,8.999999E+09,8.999999E+09,8.999999E+09,8.999999E+09]];
	LOCAL CONST Robtarget Tr_meulage_bavure_P2 :=[[108.60534375,-130.8681796875,116.9267109375],[0.491094715245722,-0.475810707049947,-0.507741056989115,0.524050733003905],[0,0,0,0],[8.999999E+09,8.999999E+09,8.999999E+09,8.999999E+09,8.999999E+09,8.999999E+09]];
	LOCAL CONST Robtarget Tr_meulage_bavure_P3 :=[[108.5476953125,-130.21634375,116.837421875],[0.492570509269526,-0.47700414491286,-0.506375695076233,0.522900558968886],[0,0,0,0],[8.999999E+09,8.999999E+09,8.999999E+09,8.999999E+09,8.999999E+09,8.999999E+09]];
	LOCAL CONST Robtarget Tr_meulage_bavure_P4 :=[[108.42959375,-126.9828984375,116.3944921875],[0.494344435998688,-0.478396808891374,-0.504724060485934,0.521549321355403],[0,0,0,0],[8.999999E+09,8.999999E+09,8.999999E+09,8.999999E+09,8.999999E+09,8.999999E+09]];
	LOCAL CONST Robtarget Tr_meulage_bavure_P5 :=[[107.94009375,-113.7517421875,114.5820546875],[0.496199764240407,-0.479790103164328,-0.50298395265102,0.520186883964681],[0,0,0,0],[8.999999E+09,8.999999E+09,8.999999E+09,8.999999E+09,8.999999E+09,8.999999E+09]];
	LOCAL CONST Robtarget Tr_meulage_bavure_P6 :=[[107.861234375,-110.992390625,114.2040625],[0.497966802776015,-0.481036814703158,-0.501313946206237,0.518957583596582],[0,0,0,0],[8.999999E+09,8.999999E+09,8.999999E+09,8.999999E+09,8.999999E+09,8.999999E+09]];
	LOCAL CONST Robtarget Tr_meulage_bavure_P7 :=[[107.83978125,-109.450546875,113.992859375],[0.499534079012983,-0.482040548102463,-0.499820630436831,0.517959410841677],[0,0,0,0],[8.999999E+09,8.999999E+09,8.999999E+09,8.999999E+09,8.999999E+09,8.999999E+09]];
	LOCAL CONST Robtarget Tr_meulage_bavure_P8 :=[[107.728390625,-107.482484375,113.723265625],[0.500830965913334,-0.482749596308721,-0.498573791959862,0.517247856270906],[0,0,0,0],[8.999999E+09,8.999999E+09,8.999999E+09,8.999999E+09,8.999999E+09,8.999999E+09]];
	LOCAL CONST Robtarget Tr_meulage_bavure_P9 :=[[107.6213046875,-103.8069921875,113.2197890625],[0.501803088568997,-0.483131967284052,-0.497627982534132,0.516859316922764],[0,0,0,0],[8.999999E+09,8.999999E+09,8.999999E+09,8.999999E+09,8.999999E+09,8.999999E+09]];
	LOCAL CONST Robtarget Tr_meulage_bavure_P10 :=[[107.4977734375,-98.98315625,112.5590078125],[0.502392939726944,-0.483151062660252,-0.497039608653659,0.516834608160295],[0,0,0,0],[8.999999E+09,8.999999E+09,8.999999E+09,8.999999E+09,8.999999E+09,8.999999E+09]];
	LOCAL CONST Robtarget Tr_meulage_bavure_P11 :=[[107.4833671875,-98.2393359375,112.4571171875],[0.502579255059713,-0.482801242566197,-0.496829544111376,0.517182227709192],[0,0,0,0],[8.999999E+09,8.999999E+09,8.999999E+09,8.999999E+09,8.999999E+09,8.999999E+09]];
	LOCAL CONST Robtarget Tr_meulage_bavure_P12 :=[[107.3741796875,-92.14703125,111.6225703125],[0.502395905039351,-0.482130496262875,-0.496965779709902,0.517854760497897],[0,0,0,0],[8.999999E+09,8.999999E+09,8.999999E+09,8.999999E+09,8.999999E+09,8.999999E+09]];
	LOCAL CONST Robtarget Tr_meulage_bavure_P13 :=[[107.2834765625,-85.8595546875,110.761296875],[0.501945673835336,-0.481260349882982,-0.497352126014942,0.518729099720574],[0,0,0,0],[8.999999E+09,8.999999E+09,8.999999E+09,8.999999E+09,8.999999E+09,8.999999E+09]];
	LOCAL CONST Robtarget Tr_meulage_bavure_P14 :=[[107.289765625,-84.8499921875,110.623],[0.501389083037784,-0.480357667454232,-0.497839224255455,0.519636031777231],[0,0,0,0],[8.999999E+09,8.999999E+09,8.999999E+09,8.999999E+09,8.999999E+09,8.999999E+09]];
	LOCAL CONST Robtarget Tr_meulage_bavure_P15 :=[[107.26553125,-84.582453125,110.5863515625],[0.500876738083504,-0.479569288365527,-0.498288222203907,0.520427361421631],[0,0,0,0],[8.999999E+09,8.999999E+09,8.999999E+09,8.999999E+09,8.999999E+09,8.999999E+09]];
	LOCAL CONST Robtarget Tr_meulage_bavure_P16 :=[[107.265625,-84.20575,110.53475],[0.500510314668251,-0.479001149193476,-0.498607468739846,0.520997040393572],[0,0,0,0],[8.999999E+09,8.999999E+09,8.999999E+09,8.999999E+09,8.999999E+09,8.999999E+09]];
	LOCAL CONST Robtarget Tr_meulage_bavure_P17 :=[[107.224671875,-83.3940546875,110.4235625],[0.500347300047611,-0.478715277692832,-0.498746264891374,0.521283440649561],[0,0,0,0],[8.999999E+09,8.999999E+09,8.999999E+09,8.999999E+09,8.999999E+09,8.999999E+09]];
	LOCAL CONST Robtarget Tr_meulage_bavure_P18 :=[[106.8244921875,-75.0358125,109.278625],[0.500420773952346,-0.478748501058071,-0.498675630111192,0.521249976177257],[0,0,0,0],[8.999999E+09,8.999999E+09,8.999999E+09,8.999999E+09,8.999999E+09,8.999999E+09]];
	LOCAL CONST Robtarget Tr_meulage_bavure_P19 :=[[106.7139296875,-72.9476171875,108.992578125],[0.50077525106977,-0.479137371072243,-0.498353993554007,0.520859697679482],[0,0,0,0],[8.999999E+09,8.999999E+09,8.999999E+09,8.999999E+09,8.999999E+09,8.999999E+09]];
	LOCAL CONST Robtarget Tr_meulage_bavure_P20 :=[[106.5289609375,-69.2815390625,108.490390625],[0.501437785644862,-0.47990318121429,-0.497754396458258,0.520090035084751],[0,0,0,0],[8.999999E+09,8.999999E+09,8.999999E+09,8.999999E+09,8.999999E+09,8.999999E+09]];
	LOCAL CONST Robtarget Tr_meulage_bavure_P21 :=[[106.2872890625,-64.42249609375,107.82478125],[0.502399611122831,-0.481040337900743,-0.49688177024212,0.518944438699389],[0,0,0,0],[8.999999E+09,8.999999E+09,8.999999E+09,8.999999E+09,8.999999E+09,8.999999E+09]];
	LOCAL CONST Robtarget Tr_meulage_bavure_P22 :=[[106.2378828125,-62.860890625,107.6108671875],[0.50359686112984,-0.482479646783683,-0.495790092744705,0.517489879935697],[0,0,0,0],[8.999999E+09,8.999999E+09,8.999999E+09,8.999999E+09,8.999999E+09,8.999999E+09]];
	LOCAL CONST Robtarget Tr_meulage_bavure_P23 :=[[106.2523203125,-61.49397265625,107.423625],[0.504902405352767,-0.484088772445622,-0.49459282272255,0.51585808239517],[0,0,0,0],[8.999999E+09,8.999999E+09,8.999999E+09,8.999999E+09,8.999999E+09,8.999999E+09]];
	LOCAL CONST Robtarget Tr_meulage_bavure_P24 :=[[106.1898828125,-57.68580078125,106.90196875],[0.506172529634505,-0.485730176125717,-0.49342244915574,0.514188538294503],[0,0,0,0],[8.999999E+09,8.999999E+09,8.999999E+09,8.999999E+09,8.999999E+09,8.999999E+09]];
	LOCAL CONST Robtarget Tr_meulage_bavure_P25 :=[[106.1760859375,-57.69946875,106.90384375],[0.507282288131088,-0.487274166280227,-0.492396580481455,0.512615035435527],[0,0,0,0],[8.999999E+09,8.999999E+09,8.999999E+09,8.999999E+09,8.999999E+09,8.999999E+09]];
	LOCAL CONST Robtarget Tr_meulage_bavure_P26 :=[[106.133578125,-55.0497109375,106.540875],[0.508137140749868,-0.48862372130124,-0.491607086469656,0.511239648017535],[0,0,0,0],[8.999999E+09,8.999999E+09,8.999999E+09,8.999999E+09,8.999999E+09,8.999999E+09]];
	LOCAL CONST Robtarget Tr_meulage_bavure_P27 :=[[106.1247890625,-50.14363671875,105.8688203125],[0.508690422198637,-0.489717850750097,-0.49110128027081,0.510127448326837],[0,0,0,0],[8.999999E+09,8.999999E+09,8.999999E+09,8.999999E+09,8.999999E+09,8.999999E+09]];
	LOCAL CONST Robtarget Tr_meulage_bavure_P28 :=[[106.121765625,-49.92137890625,105.838375],[0.508908636854013,-0.490520000462624,-0.490914663357534,0.509318094889723],[0,0,0,0],[8.999999E+09,8.999999E+09,8.999999E+09,8.999999E+09,8.999999E+09,8.999999E+09]];
	LOCAL CONST Robtarget Tr_meulage_bavure_P29 :=[[106.1225625,-49.7881328125,105.820125],[0.508763640879701,-0.491004509800079,-0.491077310617219,0.50883907482796],[0,0,0,0],[8.999999E+09,8.999999E+09,8.999999E+09,8.999999E+09,8.999999E+09,8.999999E+09]];
	LOCAL CONST Robtarget Tr_meulage_bavure_P30 :=[[106.043578125,-42.98191015625,104.8877890625],[0.508242887845312,-0.491141705031895,-0.491602604876488,0.508719835874004],[0,0,0,0],[8.999999E+09,8.999999E+09,8.999999E+09,8.999999E+09,8.999999E+09,8.999999E+09]];
	LOCAL CONST Robtarget Tr_meulage_bavure_P31 :=[[106.0759296875,-41.8627265625,104.7344765625],[0.507350211856743,-0.490925198052236,-0.492487069595253,0.508964339347829],[0,0,0,0],[8.999999E+09,8.999999E+09,8.999999E+09,8.999999E+09,8.999999E+09,8.999999E+09]];
	LOCAL CONST Robtarget Tr_meulage_bavure_P32 :=[[105.9424140625,-39.0018984375,104.34259375],[0.506134479285983,-0.490405045928722,-0.493682862425567,0.509517429685044],[0,0,0,0],[8.999999E+09,8.999999E+09,8.999999E+09,8.999999E+09,8.999999E+09,8.999999E+09]];
	LOCAL CONST Robtarget Tr_meulage_bavure_P33 :=[[105.9767734375,-36.497484375,103.99953125],[0.504702751494391,-0.489671839649961,-0.495084838505319,0.510281907155228],[0,0,0,0],[8.999999E+09,8.999999E+09,8.999999E+09,8.999999E+09,8.999999E+09,8.999999E+09]];
	LOCAL CONST Robtarget Tr_meulage_bavure_P34 :=[[105.9813828125,-33.15996875,103.5423515625],[0.503203893093163,-0.488866256649437,-0.496548648706148,0.511111596966407],[0,0,0,0],[8.999999E+09,8.999999E+09,8.999999E+09,8.999999E+09,8.999999E+09,8.999999E+09]];
	LOCAL CONST Robtarget Tr_meulage_bavure_P35 :=[[105.9880703125,-32.419296875,103.440890625],[0.501799688523473,-0.488140707355646,-0.497919164865827,0.51185176338408],[0,0,0,0],[8.999999E+09,8.999999E+09,8.999999E+09,8.999999E+09,8.999999E+09,8.999999E+09]];
	LOCAL CONST Robtarget Tr_meulage_bavure_P36 :=[[105.710265625,-26.42346875,102.6195625],[0.500617314213888,-0.487614980125734,-0.499075890715883,0.51238383188036],[0,0,0,0],[8.999999E+09,8.999999E+09,8.999999E+09,8.999999E+09,8.999999E+09,8.999999E+09]];
	LOCAL CONST Robtarget Tr_meulage_bavure_P37 :=[[105.50121875,-20.493767578125,101.807296875],[0.499720879057156,-0.487345998104937,-0.499958822835919,0.512653973586442],[0,0,0,0],[8.999999E+09,8.999999E+09,8.999999E+09,8.999999E+09,8.999999E+09,8.999999E+09]];
	LOCAL CONST Robtarget Tr_meulage_bavure_P38 :=[[105.3786953125,-19.161875,101.6248515625],[0.499121970261473,-0.487337059022142,-0.500557304245155,0.512661910885505],[0,0,0,0],[8.999999E+09,8.999999E+09,8.999999E+09,8.999999E+09,8.999999E+09,8.999999E+09]];
	LOCAL CONST Robtarget Tr_meulage_bavure_P39 :=[[105.150421875,-12.1058818359375,100.658296875],[0.498804358088272,-0.487572629988022,-0.500886769047871,0.512425201791925],[0,0,0,0],[8.999999E+09,8.999999E+09,8.999999E+09,8.999999E+09,8.999999E+09,8.999999E+09]];
	LOCAL CONST Robtarget Tr_meulage_bavure_P40 :=[[105.1194765625,-11.0708388671875,100.516515625],[0.498757570857914,-0.488036137379024,-0.500956177983542,0.511961445681409],[0,0,0,0],[8.999999E+09,8.999999E+09,8.999999E+09,8.999999E+09,8.999999E+09,8.999999E+09]];
	LOCAL CONST Robtarget Tr_meulage_bavure_P41 :=[[104.988375,-4.15126611328125,99.56865625],[0.498980404329158,-0.488717803399697,-0.500765023278066,0.511280604166639],[0,0,0,0],[8.999999E+09,8.999999E+09,8.999999E+09,8.999999E+09,8.999999E+09,8.999999E+09]];
	LOCAL CONST Robtarget Tr_meulage_bavure_P42 :=[[104.9229765625,-1.61788684082031,99.221625],[0.49944900060102,-0.489590984012762,-0.500334288847441,0.510408624119522],[0,0,0,0],[8.999999E+09,8.999999E+09,8.999999E+09,8.999999E+09,8.999999E+09,8.999999E+09]];
	LOCAL CONST Robtarget Tr_meulage_bavure_P43 :=[[104.8765234375,-0.663028259277344,99.0908203125],[0.5000843887141,-0.490573511680102,-0.499737879259299,0.509426428285495],[0,0,0,0],[8.999999E+09,8.999999E+09,8.999999E+09,8.999999E+09,8.999999E+09,8.999999E+09]];
	LOCAL CONST Robtarget Tr_meulage_bavure_P44 :=[[104.4556875,8.1892099609375,97.87821875],[0.500729325048277,-0.49151022188555,-0.499126533707428,0.508488493643584],[0,0,0,0],[8.999999E+09,8.999999E+09,8.999999E+09,8.999999E+09,8.999999E+09,8.999999E+09]];
	LOCAL CONST Robtarget Tr_meulage_bavure_P45 :=[[104.3269375,10.6936240234375,97.53515625],[0.501188805678061,-0.492204985488596,-0.498689711119147,0.507791891769721],[0,0,0,0],[8.999999E+09,8.999999E+09,8.999999E+09,8.999999E+09,8.999999E+09,8.999999E+09]];
	LOCAL CONST Robtarget Tr_meulage_bavure_P46 :=[[104.3324296875,12.6696171875,97.2644765625],[0.501288394661472,-0.492485276757993,-0.498598711193225,0.507511106036885],[0,0,0,0],[8.999999E+09,8.999999E+09,8.999999E+09,8.999999E+09,8.999999E+09,8.999999E+09]];
	LOCAL CONST Robtarget Tr_meulage_bavure_P47 :=[[104.3413125,13.4405244140625,97.158875],[0.500939012221703,-0.492265281023728,-0.498941359731908,0.507732723666546],[0,0,0,0],[8.999999E+09,8.999999E+09,8.999999E+09,8.999999E+09,8.999999E+09,8.999999E+09]];
	LOCAL CONST Robtarget Tr_meulage_bavure_P48 :=[[104.3224453125,14.54311328125,97.00784375],[0.500181814866547,-0.491587288341717,-0.499676629826626,0.508412584052313],[0,0,0,0],[8.999999E+09,8.999999E+09,8.999999E+09,8.999999E+09,8.999999E+09,8.999999E+09]];
	LOCAL CONST Robtarget Tr_meulage_bavure_P49 :=[[104.2218359375,16.480494140625,96.742453125],[0.499175364189146,-0.490613465727521,-0.500648426602098,0.509385449315454],[0,0,0,0],[8.999999E+09,8.999999E+09,8.999999E+09,8.999999E+09,8.999999E+09,8.999999E+09]];
	LOCAL CONST Robtarget Tr_meulage_bavure_P50 :=[[104.267484375,18.432693359375,96.47503125],[0.498144888299916,-0.489566356065362,-0.501637493424126,0.510427544770761],[0,0,0,0],[8.999999E+09,8.999999E+09,8.999999E+09,8.999999E+09,8.999999E+09,8.999999E+09]];
	LOCAL CONST Robtarget Tr_meulage_bavure_P51 :=[[104.214359375,19.989896484375,96.2617265625],[0.497304743380418,-0.488665622564939,-0.502438586103878,0.511321199177673],[0,0,0,0],[8.999999E+09,8.999999E+09,8.999999E+09,8.999999E+09,8.999999E+09,8.999999E+09]];
	LOCAL CONST Robtarget Tr_meulage_bavure_P52 :=[[103.8442109375,27.250796875,95.2671015625],[0.496800672704333,-0.488063739094321,-0.502914784199545,0.511917569551308],[0,0,0,0],[8.999999E+09,8.999999E+09,8.999999E+09,8.999999E+09,8.999999E+09,8.999999E+09]];
	LOCAL CONST Robtarget Tr_meulage_bavure_P53 :=[[103.74884375,30.07655078125,94.8800234375],[0.49668656083056,-0.487816368433426,-0.503017001532339,0.512163594126085],[0,0,0,0],[8.999999E+09,8.999999E+09,8.999999E+09,8.999999E+09,8.999999E+09,8.999999E+09]];
	LOCAL CONST Robtarget Tr_meulage_bavure_P54 :=[[103.702453125,31.465798828125,94.68971875],[0.496922035013948,-0.487892998195233,-0.502785179190606,0.512089813427229],[0,0,0,0],[8.999999E+09,8.999999E+09,8.999999E+09,8.999999E+09,8.999999E+09,8.999999E+09]];
	LOCAL CONST Robtarget Tr_meulage_bavure_P55 :=[[103.5766875,35.095328125,94.1925390625],[0.497398351136741,-0.488189700650875,-0.502322930025156,0.511798173536993],[0,0,0,0],[8.999999E+09,8.999999E+09,8.999999E+09,8.999999E+09,8.999999E+09,8.999999E+09]];
	LOCAL CONST Robtarget Tr_meulage_bavure_P56 :=[[103.36340625,39.8841015625,93.5365546875],[0.497979225004435,-0.488572770635122,-0.501759741080758,0.511420083188442],[0,0,0,0],[8.999999E+09,8.999999E+09,8.999999E+09,8.999999E+09,8.999999E+09,8.999999E+09]];
	LOCAL CONST Robtarget Tr_meulage_bavure_P57 :=[[103.29565625,41.5240625,93.3119140625],[0.498529822445976,-0.488916125390866,-0.501224523306461,0.51108024389618],[0,0,0,0],[8.999999E+09,8.999999E+09,8.999999E+09,8.999999E+09,8.999999E+09,8.999999E+09]];
	LOCAL CONST Robtarget Tr_meulage_bavure_P58 :=[[103.323546875,44.598078125,92.8908203125],[0.498953339217476,-0.48912792500005,-0.500810266299137,0.51087035090937],[0,0,0,0],[8.999999E+09,8.999999E+09,8.999999E+09,8.999999E+09,8.999999E+09,8.999999E+09]];
	LOCAL CONST Robtarget Tr_meulage_bavure_P59 :=[[103.214265625,49.24574609375,92.254171875],[0.499218812661837,-0.489170881319766,-0.500546639301685,0.510828237118053],[0,0,0,0],[8.999999E+09,8.999999E+09,8.999999E+09,8.999999E+09,8.999999E+09,8.999999E+09]];
	LOCAL CONST Robtarget Tr_meulage_bavure_P60 :=[[102.758546875,59.68599609375,90.8240390625],[0.499367318609649,-0.489080685219213,-0.500394201597639,0.510918787536312],[0,0,0,0],[8.999999E+09,8.999999E+09,8.999999E+09,8.999999E+09,8.999999E+09,8.999999E+09]];
	LOCAL CONST Robtarget Tr_meulage_bavure_P61 :=[[102.7488984375,60.20791796875,90.7525390625],[0.499498215569915,-0.488956673824385,-0.500257850944735,0.511043037652622],[0,0,0,0],[8.999999E+09,8.999999E+09,8.999999E+09,8.999999E+09,8.999999E+09,8.999999E+09]];
	LOCAL CONST Robtarget Tr_meulage_bavure_P62 :=[[102.7326328125,60.58253125,90.7012265625],[0.499755640663383,-0.488940546646473,-0.499999707051082,0.511059423569326],[0,0,0,0],[8.999999E+09,8.999999E+09,8.999999E+09,8.999999E+09,8.999999E+09,8.999999E+09]];
	LOCAL CONST Robtarget Tr_meulage_bavure_P63 :=[[102.5277734375,68.640671875,89.5973984375],[0.500299733116974,-0.489182222868727,-0.499466198400793,0.510817429741151],[0,0,0,0],[8.999999E+09,8.999999E+09,8.999999E+09,8.999999E+09,8.999999E+09,8.999999E+09]];
	LOCAL CONST Robtarget Tr_meulage_bavure_P64 :=[[102.49084375,69.995359375,89.411828125],[0.501253863974478,-0.489801782865865,-0.498538182342169,0.510194529663973],[0,0,0,0],[8.999999E+09,8.999999E+09,8.999999E+09,8.999999E+09,8.999999E+09,8.999999E+09]];
	LOCAL CONST Robtarget Tr_meulage_bavure_P65 :=[[102.48703125,70.0153125,89.40909375],[0.50265599177569,-0.490838905837392,-0.497176417846444,0.50914608118469],[0,0,0,0],[8.999999E+09,8.999999E+09,8.999999E+09,8.999999E+09,8.999999E+09,8.999999E+09]];
	LOCAL CONST Robtarget Tr_meulage_bavure_P66 :=[[102.4847109375,70.1021796875,89.3971953125],[0.504413904493557,-0.492204698023896,-0.49546517818648,0.507755261323218],[0,0,0,0],[8.999999E+09,8.999999E+09,8.999999E+09,8.999999E+09,8.999999E+09,8.999999E+09]];
	LOCAL CONST Robtarget Tr_meulage_bavure_P67 :=[[102.4818125,70.2071328125,89.3828203125],[0.506298183058816,-0.493680503914032,-0.493622953883251,0.50623916214187],[0,0,0,0],[8.999999E+09,8.999999E+09,8.999999E+09,8.999999E+09,8.999999E+09,8.999999E+09]];
	LOCAL CONST Robtarget Tr_meulage_bavure_P68 :=[[102.1853671875,77.40078125,88.3974140625],[0.507993624343936,-0.494966848538549,-0.491956995417499,0.504904556459451],[0,0,0,0],[8.999999E+09,8.999999E+09,8.999999E+09,8.999999E+09,8.999999E+09,8.999999E+09]];
	LOCAL CONST Robtarget Tr_meulage_bavure_P69 :=[[102.2940390625,79.5428046875,88.1039921875],[0.509203317233816,-0.495785777839736,-0.490762581603609,0.504044177337351],[0,0,0,0],[8.999999E+09,8.999999E+09,8.999999E+09,8.999999E+09,8.999999E+09,8.999999E+09]];
	LOCAL CONST Robtarget Tr_meulage_bavure_P70 :=[[102.340578125,81.494640625,87.836625],[0.509761271361685,-0.495981986300854,-0.490207957383415,0.503826829379657],[0,0,0,0],[8.999999E+09,8.999999E+09,8.999999E+09,8.999999E+09,8.999999E+09,8.999999E+09]];
	LOCAL CONST Robtarget Tr_meulage_bavure_P71 :=[[102.3500703125,84.57315625,87.414921875],[0.509688925859904,-0.495585566334941,-0.490273745403746,0.504225941284297],[0,0,0,0],[8.999999E+09,8.999999E+09,8.999999E+09,8.999999E+09,8.999999E+09,8.999999E+09]];
	LOCAL CONST Robtarget Tr_meulage_bavure_P72 :=[[102.23175,87.872546875,86.9629609375],[0.50916444456345,-0.494785379385685,-0.490782917309748,0.505045666069406],[0,0,0,0],[8.999999E+09,8.999999E+09,8.999999E+09,8.999999E+09,8.999999E+09,8.999999E+09]];
	LOCAL CONST Robtarget Tr_meulage_bavure_P73 :=[[102.210296875,88.715171875,86.84753125],[0.508438153473989,-0.493835319235846,-0.491487598242562,0.506021009782152],[0,0,0,0],[8.999999E+09,8.999999E+09,8.999999E+09,8.999999E+09,8.999999E+09,8.999999E+09]];
	LOCAL CONST Robtarget Tr_meulage_bavure_P74 :=[[102.19659375,89.406984375,86.752765625],[0.507725505516407,-0.492942920094182,-0.492176583915375,0.506936188116929],[0,0,0,0],[8.999999E+09,8.999999E+09,8.999999E+09,8.999999E+09,8.999999E+09,8.999999E+09]];
	LOCAL CONST Robtarget Tr_meulage_bavure_P75 :=[[102.1690078125,92.3888359375,86.3443046875],[0.507135447933651,-0.492213787870748,-0.492744901861548,0.5076826628599],[0,0,0,0],[8.999999E+09,8.999999E+09,8.999999E+09,8.999999E+09,8.999999E+09,8.999999E+09]];
	LOCAL CONST Robtarget Tr_meulage_bavure_P76 :=[[102.057859375,96.6589921875,85.7593671875],[0.5066699779413,-0.491644774633008,-0.493191906679407,0.508264392039175],[0,0,0,0],[8.999999E+09,8.999999E+09,8.999999E+09,8.999999E+09,8.999999E+09,8.999999E+09]];
	LOCAL CONST Robtarget Tr_meulage_bavure_P77 :=[[102.055234375,96.7636640625,85.7450234375],[0.506272659370754,-0.491171005232566,-0.493572847189918,0.508748348900842],[0,0,0,0],[8.999999E+09,8.999999E+09,8.999999E+09,8.999999E+09,8.999999E+09,8.999999E+09]];
	LOCAL CONST Robtarget Tr_meulage_bavure_P78 :=[[102.073,100.0059375,85.300890625],[0.505889524125324,-0.490727259052295,-0.493939815467116,0.509201340630194],[0,0,0,0],[8.999999E+09,8.999999E+09,8.999999E+09,8.999999E+09,8.999999E+09,8.999999E+09]];
	LOCAL CONST Robtarget Tr_meulage_bavure_P79 :=[[102.025359375,100.9899140625,85.1661015625],[0.505504507860943,-0.490270803982556,-0.494307377813463,0.509666506191787],[0,0,0,0],[8.999999E+09,8.999999E+09,8.999999E+09,8.999999E+09,8.999999E+09,8.999999E+09]];
	LOCAL CONST Robtarget Tr_meulage_bavure_P80 :=[[102.037265625,101.6950859375,85.0695078125],[0.505133588969922,-0.489792017371884,-0.494659102216418,0.510153123686989],[0,0,0,0],[8.999999E+09,8.999999E+09,8.999999E+09,8.999999E+09,8.999999E+09,8.999999E+09]];
	LOCAL CONST Robtarget Tr_meulage_bavure_P81 :=[[101.9645078125,107.525921875,84.27078125],[0.504809665463237,-0.489295982061108,-0.494962193359731,0.510655530409957],[0,0,0,0],[8.999999E+09,8.999999E+09,8.999999E+09,8.999999E+09,8.999999E+09,8.999999E+09]];
	LOCAL CONST Robtarget Tr_meulage_bavure_P82 :=[[101.9210546875,109.6221328125,83.9836328125],[0.504560749928977,-0.488772228272319,-0.4951880781942,0.511183847275278],[0,0,0,0],[8.999999E+09,8.999999E+09,8.999999E+09,8.999999E+09,8.999999E+09,8.999999E+09]];
	LOCAL CONST Robtarget Tr_meulage_bavure_P83 :=[[101.7733125,114.9953203125,83.2476015625],[0.504358482774698,-0.488163788055874,-0.495362243534725,0.511795744965107],[0,0,0,0],[8.999999E+09,8.999999E+09,8.999999E+09,8.999999E+09,8.999999E+09,8.999999E+09]];
	LOCAL CONST Robtarget Tr_meulage_bavure_P84 :=[[101.6951015625,121.0461484375,82.4187421875],[0.504112327662326,-0.487353427960789,-0.495568672363761,0.51261007435024],[0,0,0,0],[8.999999E+09,8.999999E+09,8.999999E+09,8.999999E+09,8.999999E+09,8.999999E+09]];
	LOCAL CONST Robtarget Tr_meulage_bavure_P85 :=[[101.6745625,121.75921875,82.3210625],[0.503617094935733,-0.48611272757526,-0.495997924059393,0.513858246121055],[0,0,0,0],[8.999999E+09,8.999999E+09,8.999999E+09,8.999999E+09,8.999999E+09,8.999999E+09]];
	LOCAL CONST Robtarget Tr_meulage_bavure_P86 :=[[101.517515625,130.544265625,81.1176640625],[0.502547456017733,-0.484105899934867,-0.496947669981511,0.515878421140393],[0,0,0,0],[8.999999E+09,8.999999E+09,8.999999E+09,8.999999E+09,8.999999E+09,8.999999E+09]];
	LOCAL CONST Robtarget Tr_meulage_bavure_P87 :=[[101.6070859375,131.092125,81.042609375],[0.500480423224856,-0.480914383396575,-0.498790844209598,0.519084189263782],[0,0,0,0],[8.999999E+09,8.999999E+09,8.999999E+09,8.999999E+09,8.999999E+09,8.999999E+09]];
	LOCAL CONST Robtarget Tr_meulage_bavure_P88 :=[[101.56765625,132.701015625,80.82221875],[0.496865743862169,-0.476014913093535,-0.5019836535666,0.523971990320833],[0,0,0,0],[8.999999E+09,8.999999E+09,8.999999E+09,8.999999E+09,8.999999E+09,8.999999E+09]];
	LOCAL CONST Robtarget Tr_meulage_bavure_P89 :=[[101.5835859375,137.5764375,80.154375],[0.491104810327846,-0.468854272694611,-0.506961029765153,0.531020009555491],[0,0,0,0],[8.999999E+09,8.999999E+09,8.999999E+09,8.999999E+09,8.999999E+09,8.999999E+09]];
	LOCAL CONST Robtarget Tr_meulage_bavure_P90 :=[[101.5303984375,138.495625,80.0284609375],[0.482400213889277,-0.458710992944574,-0.514226235221522,0.54078243092882],[0,0,0,0],[8.999999E+09,8.999999E+09,8.999999E+09,8.999999E+09,8.999999E+09,8.999999E+09]];
	LOCAL CONST Robtarget Tr_meulage_bavure_P91 :=[[101.5815703125,141.553921875,79.6095234375],[0.469558837659316,-0.444511154243735,-0.524431144431496,0.553982225779137],[0,0,0,0],[8.999999E+09,8.999999E+09,8.999999E+09,8.999999E+09,8.999999E+09,8.999999E+09]];
	LOCAL CONST Robtarget Tr_meulage_bavure_P92 :=[[101.232515625,143.4361875,79.3516875],[0.45071877169164,-0.424601269757008,-0.538426078468185,0.571545018866308],[0,0,0,0],[8.999999E+09,8.999999E+09,8.999999E+09,8.999999E+09,8.999999E+09,8.999999E+09]];
	LOCAL CONST Robtarget Tr_meulage_bavure_P93 :=[[100.9292890625,144.95534375,79.1435859375],[0.423087637340002,-0.396510194804103,-0.557123243973814,0.594466321645357],[0,0,0,0],[8.999999E+09,8.999999E+09,8.999999E+09,8.999999E+09,8.999999E+09,8.999999E+09]];
	LOCAL CONST Robtarget Tr_meulage_bavure_P94 :=[[100.3225390625,145.76253125,79.033015625],[0.38316130186514,-0.357133253646006,-0.580809955558974,0.623139672478659],[0,0,0,0],[8.999999E+09,8.999999E+09,8.999999E+09,8.999999E+09,8.999999E+09,8.999999E+09]];
	LOCAL CONST Robtarget Tr_meulage_bavure_P95 :=[[99.5499609375,147.1056875,78.84903125],[0.327946967023897,-0.303945942719956,-0.608020428853117,0.656032627863261],[0,0,0,0],[8.999999E+09,8.999999E+09,8.999999E+09,8.999999E+09,8.999999E+09,8.999999E+09]];
	LOCAL CONST Robtarget Tr_meulage_bavure_P96 :=[[98.1312578125,147.94725,78.73375],[0.258327309872839,-0.238056225543317,-0.634475910768032,0.688503124981294],[0,0,0,0],[8.999999E+09,8.999999E+09,8.999999E+09,8.999999E+09,8.999999E+09,8.999999E+09]];
	LOCAL CONST Robtarget Tr_meulage_bavure_P97 :=[[96.994875,148.377046875,78.674875],[0.182318581427254,-0.167056767010562,-0.65459307099266,0.714394766827649],[0,0,0,0],[8.999999E+09,8.999999E+09,8.999999E+09,8.999999E+09,8.999999E+09,8.999999E+09]];
	LOCAL CONST Robtarget Tr_meulage_bavure_P98 :=[[95.629515625,148.31496875,78.683375],[0.112248848095117,-0.102279808211857,-0.66570974850354,0.730595351532446],[0,0,0,0],[8.999999E+09,8.999999E+09,8.999999E+09,8.999999E+09,8.999999E+09,8.999999E+09]];
	LOCAL CONST Robtarget Tr_meulage_bavure_P99 :=[[93.6759375,148.418125,78.6692421875],[0.056957146386199,-0.0516209727188796,-0.669557878785362,0.738771551704276],[0,0,0,0],[8.999999E+09,8.999999E+09,8.999999E+09,8.999999E+09,8.999999E+09,8.999999E+09]];
	LOCAL CONST Robtarget Tr_meulage_bavure_P100 :=[[89.6470625,147.91253125,78.7385],[0.0185843106977833,-0.0167578812345148,-0.669461259592401,0.742425362388284],[0,0,0,0],[8.999999E+09,8.999999E+09,8.999999E+09,8.999999E+09,8.999999E+09,8.999999E+09]];
	LOCAL CONST Robtarget Tr_meulage_bavure_P101 :=[[87.43734375,147.60353125,78.780828125],[0.00502796121181569,-0.00451243886079119,0.667908106685,-0.744213086774238],[0,0,0,0],[8.999999E+09,8.999999E+09,8.999999E+09,8.999999E+09,8.999999E+09,8.999999E+09]];
	LOCAL CONST Robtarget Tr_meulage_bavure_P102 :=[[86.649875,147.523734375,78.791765625],[0.0174341232496472,-0.0155788610294561,0.666135323949124,-0.745464338934289],[0,0,0,0],[8.999999E+09,8.999999E+09,8.999999E+09,8.999999E+09,8.999999E+09,8.999999E+09]];
	LOCAL CONST Robtarget Tr_meulage_bavure_P103 :=[[83.978671875,147.320796875,78.8195625],[0.0222999297998446,-0.0198502151461422,0.664592242979521,-0.746609558377753],[0,0,0,0],[8.999999E+09,8.999999E+09,8.999999E+09,8.999999E+09,8.999999E+09,8.999999E+09]];
	LOCAL CONST Robtarget Tr_meulage_bavure_P104 :=[[75.878234375,147.023109375,78.8603359375],[0.0227904214257368,-0.0202187905002687,0.663333736084847,-0.747703251145574],[0,0,0,0],[8.999999E+09,8.999999E+09,8.999999E+09,8.999999E+09,8.999999E+09,8.999999E+09]];
	LOCAL CONST Robtarget Tr_meulage_bavure_P105 :=[[67.2933359375,146.72353125,78.901375],[0.0213168071843018,-0.018856857027962,0.662299212868805,-0.74869871464285],[0,0,0,0],[8.999999E+09,8.999999E+09,8.999999E+09,8.999999E+09,8.999999E+09,8.999999E+09]];
	LOCAL CONST Robtarget Tr_meulage_bavure_P106 :=[[64.1331171875,146.56171875,78.9235390625],[0.0194229180624858,-0.0171402056646551,0.661450315362452,-0.749541489118931],[0,0,0,0],[8.999999E+09,8.999999E+09,8.999999E+09,8.999999E+09,8.999999E+09,8.999999E+09]];
	LOCAL CONST Robtarget Tr_meulage_bavure_P107 :=[[43.76840234375,145.79140625,79.0290625],[0.0178297843938631,-0.0157039899629441,0.660768097006021,-0.750213973121505],[0,0,0,0],[8.999999E+09,8.999999E+09,8.999999E+09,8.999999E+09,8.999999E+09,8.999999E+09]];
	LOCAL CONST Robtarget Tr_meulage_bavure_P108 :=[[29.889892578125,145.29796875,79.09665625],[0.0167328551542707,-0.0147166306129413,0.660254422748497,-0.750711349043583],[0,0,0,0],[8.999999E+09,8.999999E+09,8.999999E+09,8.999999E+09,8.999999E+09,8.999999E+09]];
	LOCAL CONST Robtarget Tr_meulage_bavure_P109 :=[[14.6651611328125,144.7896875,79.16628125],[0.015955697249741,-0.0140187981356738,0.65988932910715,-0.751062555553544],[0,0,0,0],[8.999999E+09,8.999999E+09,8.999999E+09,8.999999E+09,8.999999E+09,8.999999E+09]];
	LOCAL CONST Robtarget Tr_meulage_bavure_P110 :=[[4.66363525390625,144.41665625,79.2173828125],[0.0152076110033514,-0.0133527655689954,0.659658825339235,-0.751292663594748],[0,0,0,0],[8.999999E+09,8.999999E+09,8.999999E+09,8.999999E+09,8.999999E+09,8.999999E+09]];
	LOCAL CONST Robtarget Tr_meulage_bavure_P111 :=[[2.69107055664063,144.316421875,79.231109375],[0.014230097783162,-0.0124909301145273,0.6595698787099,-0.751404721891314],[0,0,0,0],[8.999999E+09,8.999999E+09,8.999999E+09,8.999999E+09,8.999999E+09,8.999999E+09]];
	LOCAL CONST Robtarget Tr_meulage_bavure_P112 :=[[1.34451293945313,144.240953125,79.2414453125],[0.0128510994462646,-0.0112811217905086,0.65961322552411,-0.751410658859621],[0,0,0,0],[8.999999E+09,8.999999E+09,8.999999E+09,8.999999E+09,8.999999E+09,8.999999E+09]];
	LOCAL CONST Robtarget Tr_meulage_bavure_P113 :=[[-5.1064150390625,143.969703125,79.2786015625],[0.0110383792315621,-0.00969345205529768,0.659776731808299,-0.751318078669448],[0,0,0,0],[8.999999E+09,8.999999E+09,8.999999E+09,8.999999E+09,8.999999E+09,8.999999E+09]];
	LOCAL CONST Robtarget Tr_meulage_bavure_P114 :=[[-8.497162109375,143.895453125,79.2887734375],[0.00895620543443396,-0.00787016321097035,0.660046791488863,-0.75112986890451],[0,0,0,0],[8.999999E+09,8.999999E+09,8.999999E+09,8.999999E+09,8.999999E+09,8.999999E+09]];
	LOCAL CONST Robtarget Tr_meulage_bavure_P115 :=[[-25.929138671875,143.37446875,79.360140625],[0.00694342048117971,-0.00610710795748403,0.660410578362354,-0.750847760955254],[0,0,0,0],[8.999999E+09,8.999999E+09,8.999999E+09,8.999999E+09,8.999999E+09,8.999999E+09]];
	LOCAL CONST Robtarget Tr_meulage_bavure_P116 :=[[-32.599548828125,143.15078125,79.39078125],[0.00551359041490492,-0.00485552189432318,0.660883278981971,-0.750452740543939],[0,0,0,0],[8.999999E+09,8.999999E+09,8.999999E+09,8.999999E+09,8.999999E+09,8.999999E+09]];
	LOCAL CONST Robtarget Tr_meulage_bavure_P117 :=[[-47.24954296875,143.07553125,79.4010859375],[0.00535866404077262,-0.00472621357953622,0.661445828358821,-0.749958908055376],[0,0,0,0],[8.999999E+09,8.999999E+09,8.999999E+09,8.999999E+09,8.999999E+09,8.999999E+09]];
	LOCAL CONST Robtarget Tr_meulage_bavure_P118 :=[[-47.37057421875,143.073140625,79.401421875],[0.00724602884539085,-0.00640244956761965,0.662107737730662,-0.749346279995231],[0,0,0,0],[8.999999E+09,8.999999E+09,8.999999E+09,8.999999E+09,8.999999E+09,8.999999E+09]];
	LOCAL CONST Robtarget Tr_meulage_bavure_P119 :=[[-47.42391796875,143.07484375,79.4011875],[0.0118923880289236,-0.0105307061421585,0.662861572741511,-0.748573450449432],[0,0,0,0],[8.999999E+09,8.999999E+09,8.999999E+09,8.999999E+09,8.999999E+09,8.999999E+09]];
	LOCAL CONST Robtarget Tr_meulage_bavure_P120 :=[[-53.04476953125,143.15678125,79.3899609375],[0.020021316073296,-0.0177728261021381,0.663627059523433,-0.747584376123069],[0,0,0,0],[8.999999E+09,8.999999E+09,8.999999E+09,8.999999E+09,8.999999E+09,8.999999E+09]];
	LOCAL CONST Robtarget Tr_meulage_bavure_P121 :=[[-54.21148828125,143.1503125,79.39084375],[0.0324273228975976,-0.0288659896835659,0.664273378082254,-0.746227915948254],[0,0,0,0],[8.999999E+09,8.999999E+09,8.999999E+09,8.999999E+09,8.999999E+09,8.999999E+09]];
	LOCAL CONST Robtarget Tr_meulage_bavure_P122 :=[[-55.77984765625,142.977359375,79.4145390625],[0.0503793041707474,-0.0449858787945929,0.664530729534103,-0.744202328621204],[0,0,0,0],[8.999999E+09,8.999999E+09,8.999999E+09,8.999999E+09,8.999999E+09,8.999999E+09]];
	LOCAL CONST Robtarget Tr_meulage_bavure_P123 :=[[-57.39532421875,142.89196875,79.426234375],[0.0761518667757263,-0.0682317373885915,0.663817915861818,-0.740871849769161],[0,0,0,0],[8.999999E+09,8.999999E+09,8.999999E+09,8.999999E+09,8.999999E+09,8.999999E+09]];
	LOCAL CONST Robtarget Tr_meulage_bavure_P124 :=[[-57.56396484375,142.86509375,79.4299140625],[0.113339705773086,-0.101924605067649,0.660856846223305,-0.734869862476929],[0,0,0,0],[8.999999E+09,8.999999E+09,8.999999E+09,8.999999E+09,8.999999E+09,8.999999E+09]];
	LOCAL CONST Robtarget Tr_meulage_bavure_P125 :=[[-57.73718359375,142.79590625,79.439390625],[0.166392999801539,-0.150206340579308,0.653027344344778,-0.723399414158475],[0,0,0,0],[8.999999E+09,8.999999E+09,8.999999E+09,8.999999E+09,8.999999E+09,8.999999E+09]];
	LOCAL CONST Robtarget Tr_meulage_bavure_P126 :=[[-60.13519140625,141.812578125,79.57409375],[0.237397208297027,-0.215146246972755,0.636130490180382,-0.701920691651972],[0,0,0,0],[8.999999E+09,8.999999E+09,8.999999E+09,8.999999E+09,8.999999E+09,8.999999E+09]];
	LOCAL CONST Robtarget Tr_meulage_bavure_P127 :=[[-60.388,141.498953125,79.6170546875],[0.319651352721831,-0.290824729420739,0.606882297915686,-0.667036630131385],[0,0,0,0],[8.999999E+09,8.999999E+09,8.999999E+09,8.999999E+09,8.999999E+09,8.999999E+09]];
	LOCAL CONST Robtarget Tr_meulage_bavure_P128 :=[[-62.0285625,139.009734375,79.95803125],[0.396216173024979,-0.361847867566531,0.569053753922901,-0.623102471602584],[0,0,0,0],[8.999999E+09,8.999999E+09,8.999999E+09,8.999999E+09,8.999999E+09,8.999999E+09]];
	LOCAL CONST Robtarget Tr_meulage_bavure_P129 :=[[-62.500671875,137.096125,80.2201640625],[0.453083242870778,-0.415234830757445,0.532986401346128,-0.581567800291281],[0,0,0,0],[8.999999E+09,8.999999E+09,8.999999E+09,8.999999E+09,8.999999E+09,8.999999E+09]];
	LOCAL CONST Robtarget Tr_meulage_bavure_P130 :=[[-62.67715625,136.075875,80.359921875],[0.488638194275714,-0.449199022844039,0.506202680859215,-0.550646709662261],[0,0,0,0],[8.999999E+09,8.999999E+09,8.999999E+09,8.999999E+09,8.999999E+09,8.999999E+09]];
	LOCAL CONST Robtarget Tr_meulage_bavure_P131 :=[[-62.04891796875,131.221453125,81.0248984375],[0.508020023095603,-0.46819607450903,0.489965322891868,-0.531640926106847],[0,0,0,0],[8.999999E+09,8.999999E+09,8.999999E+09,8.999999E+09,8.999999E+09,8.999999E+09]];
	LOCAL CONST Robtarget Tr_meulage_bavure_P132 :=[[-61.806578125,129.7002265625,81.23328125],[0.51659916623023,-0.476979616328687,0.482367235501287,-0.522434299383201],[0,0,0,0],[8.999999E+09,8.999999E+09,8.999999E+09,8.999999E+09,8.999999E+09,8.999999E+09]];
	LOCAL CONST Robtarget Tr_meulage_bavure_P133 :=[[-61.6599140625,128.408546875,81.41021875],[0.518238056674101,-0.478987578502539,0.480907584091498,-0.520315396483906],[0,0,0,0],[8.999999E+09,8.999999E+09,8.999999E+09,8.999999E+09,8.999999E+09,8.999999E+09]];
	LOCAL CONST Robtarget Tr_meulage_bavure_P134 :=[[-61.60262890625,127.0141875,81.60121875],[0.515287452427863,-0.476340114842832,0.483615978939499,-0.523158218205841],[0,0,0,0],[8.999999E+09,8.999999E+09,8.999999E+09,8.999999E+09,8.999999E+09,8.999999E+09]];
	LOCAL CONST Robtarget Tr_meulage_bavure_P135 :=[[-61.4834609375,125.355296875,81.8284609375],[0.508917688226449,-0.470090380884873,0.489303048104248,-0.529717233555464],[0,0,0,0],[8.999999E+09,8.999999E+09,8.999999E+09,8.999999E+09,8.999999E+09,8.999999E+09]];
	LOCAL CONST Robtarget Tr_meulage_bavure_P136 :=[[-61.478453125,123.7001953125,82.0551796875],[0.499360308489187,-0.460504754675309,0.497515195925841,-0.539493543103056],[0,0,0,0],[8.999999E+09,8.999999E+09,8.999999E+09,8.999999E+09,8.999999E+09,8.999999E+09]];
